C01786=1116.093,234.514,-69.767,-178.654,9.768,149.567
C01787=1116.097,234.266,-69.740,-178.657,9.765,149.567
C01788=1116.102,234.018,-69.713,-178.659,9.763,149.567
C01789=1116.106,233.768,-69.685,-178.662,9.761,149.567
C01790=1116.111,233.520,-69.658,-178.665,9.758,149.567
C01791=1116.115,233.272,-69.630,-178.667,9.755,149.567
C01792=1116.120,233.023,-69.603,-178.670,9.752,149.567
C01793=1116.124,232.774,-69.576,-178.673,9.749,149.567
C01794=1116.128,232.526,-69.549,-178.676,9.746,149.567
C01795=1116.132,232.278,-69.522,-178.680,9.743,149.568
C01796=1116.137,232.030,-69.495,-178.683,9.740,149.568
C01797=1116.141,231.781,-69.467,-178.685,9.737,149.568
C01798=1116.145,231.532,-69.440,-178.688,9.734,149.568
C01799=1116.150,231.284,-69.413,-178.691,9.732,149.568
C01800=1116.154,231.036,-69.386,-178.694,9.729,149.568
C01801=1116.158,230.787,-69.359,-178.697,9.726,149.568
C01802=1116.163,230.539,-69.332,-178.700,9.722,149.568
C01803=1116.167,230.290,-69.304,-178.703,9.719,149.568
C01804=1116.172,230.041,-69.277,-178.706,9.717,149.568
C01805=1116.176,229.793,-69.251,-178.710,9.713,149.568
C01806=1116.180,229.545,-69.224,-178.713,9.710,149.568
C01807=1116.185,229.296,-69.197,-178.715,9.707,149.568
C01808=1116.189,229.048,-69.170,-178.718,9.705,149.569
C01809=1116.193,228.799,-69.143,-178.722,9.701,149.569
C01810=1116.197,228.550,-69.116,-178.724,9.698,149.569
C01811=1116.202,228.302,-69.089,-178.727,9.695,149.569
C01812=1116.207,228.053,-69.061,-178.730,9.691,149.569
C01813=1116.211,227.805,-69.035,-178.733,9.688,149.569
C01814=1116.215,227.557,-69.008,-178.736,9.685,149.569
C01815=1116.220,227.308,-68.981,-178.739,9.683,149.569
C01816=1116.224,227.060,-68.954,-178.742,9.679,149.569
C01817=1116.228,226.847,-68.931,-178.744,9.677,149.569
C01818=1116.232,226.633,-68.908,-178.747,9.674,149.569
C01819=1116.236,226.420,-68.885,-178.749,9.671,149.569
C01820=1116.239,226.207,-68.862,-178.751,9.668,149.569
C01821=1116.243,225.993,-68.840,-178.754,9.665,149.569
C01822=1116.246,225.780,-68.816,-178.756,9.663,149.569
C01823=1116.251,225.567,-68.793,-178.758,9.660,149.569
C01824=1116.254,225.354,-68.770,-178.760,9.658,149.569
C01825=1116.258,225.105,-68.744,-178.763,9.655,149.569
C01826=1116.263,224.856,-68.717,-178.766,9.651,149.569
C01827=1116.267,224.608,-68.691,-178.769,9.648,149.569
C01828=1116.271,224.359,-68.663,-178.771,9.645,149.569
C01829=1116.276,224.110,-68.636,-178.774,9.642,149.568
C01830=1116.280,223.862,-68.610,-178.777,9.639,149.568
C01831=1116.285,223.613,-68.583,-178.780,9.636,149.569
C01832=1116.289,223.365,-68.557,-178.782,9.633,149.568
C01833=1116.294,223.116,-68.530,-178.785,9.630,149.568
C01834=1116.297,222.868,-68.504,-178.787,9.627,149.568
C01835=1116.302,222.619,-68.477,-178.790,9.623,149.568
C01836=1116.306,222.370,-68.451,-178.792,9.620,149.568
C01837=1116.311,222.122,-68.424,-178.795,9.617,149.568
C01838=1116.315,221.874,-68.398,-178.797,9.614,149.568
C01839=1116.320,221.624,-68.371,-178.800,9.611,149.568
C01840=1116.324,221.376,-68.345,-178.802,9.608,149.568
C01841=1116.328,221.128,-68.318,-178.804,9.604,149.568
C01842=1116.333,220.879,-68.292,-178.807,9.601,149.568
C01843=1116.337,220.630,-68.265,-178.809,9.598,149.568
C01844=1116.342,220.382,-68.240,-178.812,9.595,149.567
C01845=1116.346,220.134,-68.213,-178.814,9.592,149.567
C01846=1116.351,219.885,-68.187,-178.817,9.589,149.567
C01847=1116.355,219.637,-68.160,-178.819,9.586,149.567
C01848=1116.360,219.388,-68.134,-178.822,9.582,149.567
C01849=1116.364,219.140,-68.108,-178.823,9.580,149.567
C01850=1116.368,218.891,-68.082,-178.826,9.577,149.567
C01851=1116.373,218.642,-68.055,-178.829,9.574,149.567
C01852=1116.377,218.393,-68.029,-178.831,9.571,149.567
C01853=1116.381,218.145,-68.002,-178.833,9.567,149.567
C01854=1116.386,217.896,-67.976,-178.836,9.564,149.566
C01855=1116.390,217.648,-67.950,-178.838,9.562,149.566
C01856=1116.394,217.399,-67.924,-178.840,9.559,149.566
C01857=1116.399,217.150,-67.898,-178.842,9.555,149.566
C01858=1116.403,216.903,-67.871,-178.844,9.553,149.566
C01859=1116.408,216.654,-67.846,-178.847,9.550,149.566
C01860=1116.412,216.405,-67.819,-178.849,9.547,149.566
C01861=1116.417,216.157,-67.793,-178.851,9.543,149.566
C01862=1116.421,215.908,-67.767,-178.853,9.541,149.566
C01863=1116.425,215.659,-67.740,-178.856,9.538,149.566
C01864=1116.430,215.410,-67.714,-178.857,9.535,149.565
C01865=1116.434,215.162,-67.689,-178.860,9.532,149.565
C01866=1116.438,214.914,-67.662,-178.862,9.529,149.565
C01867=1116.443,214.665,-67.636,-178.864,9.526,149.565
C01868=1116.448,214.416,-67.610,-178.866,9.523,149.565
C01869=1116.452,214.167,-67.585,-178.868,9.521,149.565
C01870=1116.456,213.919,-67.558,-178.871,9.517,149.565
C01871=1116.461,213.670,-67.532,-178.872,9.515,149.564
C01872=1116.466,213.422,-67.506,-178.875,9.512,149.564
C01873=1116.469,213.209,-67.484,-178.877,9.509,149.564
C01874=1116.473,212.995,-67.461,-178.879,9.506,149.564
C01875=1116.476,212.782,-67.439,-178.881,9.504,149.564
C01876=1116.480,212.568,-67.418,-178.883,9.502,149.564
C01877=1116.484,212.355,-67.395,-178.885,9.498,149.564
C01878=1116.488,212.141,-67.373,-178.888,9.497,149.564
C01879=1116.492,211.928,-67.350,-178.890,9.494,149.564
C01880=1116.495,211.714,-67.328,-178.892,9.491,149.564
C01881=1116.500,211.466,-67.303,-178.895,9.488,149.564
C01882=1116.504,211.218,-67.277,-178.898,9.485,149.564
C01883=1116.509,210.968,-67.251,-178.900,9.482,149.564
C01884=1116.513,210.720,-67.225,-178.903,9.479,149.564
C01885=1116.518,210.472,-67.200,-178.906,9.476,149.564
C01886=1116.522,210.223,-67.174,-178.907,9.474,149.564
C01887=1116.527,209.974,-67.148,-178.910,9.471,149.564
C01888=1116.531,209.725,-67.122,-178.913,9.468,149.564
C01889=1116.536,209.477,-67.097,-178.915,9.465,149.564
C01890=1116.540,209.228,-67.071,-178.918,9.462,149.564
C01891=1116.544,208.979,-67.045,-178.921,9.459,149.564
C01892=1116.548,208.731,-67.020,-178.924,9.456,149.565
C01893=1116.553,208.483,-66.994,-178.927,9.454,149.565
C01894=1116.557,208.234,-66.969,-178.929,9.450,149.565
C01895=1116.562,207.985,-66.943,-178.932,9.448,149.565
C01896=1116.566,207.737,-66.917,-178.935,9.445,149.565
C01897=1116.571,207.488,-66.892,-178.938,9.442,149.565
C01898=1116.576,207.239,-66.865,-178.941,9.439,149.565
C01899=1116.580,206.991,-66.840,-178.943,9.436,149.565
C01900=1116.584,206.742,-66.815,-178.946,9.433,149.565
C01901=1116.588,206.493,-66.790,-178.949,9.431,149.565
C01902=1116.593,206.245,-66.764,-178.952,9.427,149.565
C01903=1116.597,205.996,-66.739,-178.955,9.425,149.565
C01904=1116.602,205.747,-66.713,-178.958,9.422,149.565
C01905=1116.607,205.499,-66.687,-178.961,9.419,149.566
C01906=1116.611,205.250,-66.662,-178.963,9.416,149.566
C01907=1116.615,205.001,-66.637,-178.966,9.413,149.566
C01908=1116.620,204.753,-66.611,-178.969,9.411,149.566
C01909=1116.624,204.504,-66.586,-178.972,9.408,149.566
C01910=1116.629,204.255,-66.561,-178.975,9.404,149.566
C01911=1116.634,204.006,-66.535,-178.978,9.401,149.566
C01912=1116.638,203.758,-66.509,-178.981,9.399,149.566
C01913=1116.643,203.509,-66.484,-178.984,9.396,149.566
C01914=1116.647,203.260,-66.460,-178.986,9.393,149.566
C01915=1116.651,203.012,-66.434,-178.989,9.390,149.566
C01916=1116.656,202.763,-66.408,-178.992,9.387,149.567
C01917=1116.660,202.514,-66.383,-178.995,9.384,149.567
C01918=1116.665,202.266,-66.358,-178.998,9.381,149.567
C01919=1116.669,202.016,-66.333,-179.001,9.378,149.567
C01920=1116.674,201.769,-66.308,-179.004,9.375,149.567
C01921=1116.678,201.520,-66.282,-179.007,9.372,149.567
C01922=1116.683,201.271,-66.258,-179.010,9.369,149.567
C01923=1116.687,201.022,-66.232,-179.013,9.366,149.567
C01924=1116.691,200.773,-66.208,-179.016,9.363,149.567
C01925=1116.696,200.525,-66.182,-179.019,9.360,149.567
C01926=1116.700,200.276,-66.157,-179.022,9.357,149.567
C01927=1116.705,200.028,-66.132,-179.025,9.354,149.568
C01928=1116.709,199.778,-66.107,-179.028,9.350,149.567
C01929=1116.713,199.565,-66.086,-179.031,9.348,149.568
C01930=1116.716,199.352,-66.064,-179.033,9.345,149.568
C01931=1116.721,199.139,-66.043,-179.036,9.343,149.568
C01932=1116.724,198.925,-66.021,-179.038,9.340,149.568
C01933=1116.728,198.711,-66.000,-179.041,9.337,149.568
C01934=1116.732,198.498,-65.979,-179.043,9.334,149.568
C01935=1116.736,198.284,-65.958,-179.046,9.332,149.568
C01936=1116.740,198.071,-65.936,-179.049,9.329,149.568
C01937=1116.745,197.822,-65.911,-179.052,9.326,149.568
C01938=1116.749,197.573,-65.886,-179.055,9.322,149.568
C01939=1116.753,197.325,-65.861,-179.058,9.319,149.568
C01940=1116.758,197.076,-65.836,-179.061,9.315,149.568
C01941=1116.763,196.827,-65.811,-179.064,9.313,149.568
C01942=1116.766,196.578,-65.786,-179.067,9.309,149.568
C01943=1116.772,196.330,-65.761,-179.069,9.306,149.568
C01944=1116.775,196.080,-65.737,-179.071,9.303,149.568
C01945=1116.781,195.832,-65.712,-179.073,9.300,149.568
C01946=1116.785,195.584,-65.687,-179.075,9.298,149.568
C01947=1116.789,195.335,-65.663,-179.077,9.295,149.568
C01948=1116.794,195.086,-65.638,-179.079,9.292,149.567
C01949=1116.798,194.837,-65.613,-179.081,9.289,149.567
C01950=1116.803,194.588,-65.589,-179.083,9.287,149.567
C01951=1116.807,194.340,-65.564,-179.085,9.284,149.567
C01952=1116.812,194.091,-65.539,-179.087,9.281,149.567
C01953=1116.816,193.842,-65.515,-179.089,9.279,149.567
C01954=1116.821,193.593,-65.490,-179.091,9.275,149.567
C01955=1116.825,193.345,-65.466,-179.093,9.273,149.567
C01956=1116.830,193.096,-65.441,-179.095,9.270,149.567
C01957=1116.834,192.847,-65.417,-179.097,9.267,149.566
C01958=1116.839,192.599,-65.391,-179.099,9.265,149.566
C01959=1116.843,192.350,-65.367,-179.101,9.262,149.566
C01960=1116.848,192.101,-65.342,-179.103,9.260,149.566
C01961=1116.852,191.852,-65.318,-179.106,9.256,149.566
C01962=1116.857,191.604,-65.293,-179.107,9.254,149.566
C01963=1116.861,191.354,-65.269,-179.110,9.251,149.566
C01964=1116.866,191.106,-65.244,-179.112,9.248,149.566
C01965=1116.871,190.857,-65.220,-179.114,9.245,149.566
C01966=1116.875,190.608,-65.195,-179.116,9.243,149.566
C01967=1116.880,190.360,-65.171,-179.119,9.240,149.566
C01968=1116.884,190.111,-65.147,-179.121,9.237,149.566
C01969=1116.889,189.862,-65.122,-179.123,9.234,149.566
C01970=1116.893,189.613,-65.098,-179.125,9.232,149.566
C01971=1116.898,189.365,-65.073,-179.127,9.229,149.566
C01972=1116.902,189.115,-65.049,-179.129,9.227,149.566
C01973=1116.906,188.867,-65.025,-179.132,9.223,149.566
C01974=1116.911,188.618,-65.000,-179.134,9.220,149.566
C01975=1116.916,188.370,-64.976,-179.136,9.218,149.566
C01976=1116.920,188.121,-64.952,-179.139,9.215,149.565
C01977=1116.925,187.871,-64.928,-179.141,9.213,149.565
C01978=1116.929,187.623,-64.904,-179.143,9.209,149.565
C01979=1116.935,187.374,-64.879,-179.146,9.206,149.565
C01980=1116.938,187.125,-64.854,-179.148,9.204,149.565
C01981=1116.943,186.877,-64.830,-179.150,9.201,149.565
C01982=1116.947,186.628,-64.806,-179.153,9.198,149.565
C01983=1116.952,186.380,-64.782,-179.155,9.195,149.565
C01984=1116.956,186.130,-64.758,-179.157,9.192,149.565
C01985=1116.961,185.917,-64.737,-179.159,9.190,149.565
C01986=1116.964,185.704,-64.716,-179.162,9.187,149.565
C01987=1116.968,185.489,-64.695,-179.163,9.185,149.565
C01988=1116.972,185.276,-64.674,-179.165,9.182,149.565
C01989=1116.976,185.062,-64.655,-179.168,9.180,149.565
C01990=1116.980,184.848,-64.633,-179.170,9.177,149.565
C01991=1116.984,184.634,-64.613,-179.172,9.175,149.565
C01992=1116.987,184.422,-64.592,-179.174,9.172,149.565
C01993=1116.993,184.173,-64.568,-179.176,9.169,149.565
C01994=1116.997,183.923,-64.544,-179.179,9.166,149.565
C01995=1117.001,183.675,-64.520,-179.182,9.163,149.565
C01996=1117.006,183.426,-64.496,-179.184,9.160,149.565
C01997=1117.010,183.177,-64.472,-179.187,9.157,149.565
C01998=1117.015,182.929,-64.448,-179.189,9.154,149.565
C01999=1117.020,182.680,-64.424,-179.192,9.151,149.565
C02000=1117.024,182.430,-64.400,-179.194,9.149,149.565
C02001=1117.028,182.182,-64.376,-179.196,9.146,149.565
C02002=1117.033,181.934,-64.352,-179.199,9.143,149.565
C02003=1117.037,181.685,-64.328,-179.201,9.139,149.565
C02004=1117.042,181.436,-64.304,-179.204,9.136,149.565
C02005=1117.046,181.187,-64.281,-179.207,9.133,149.565
C02006=1117.051,180.938,-64.256,-179.210,9.129,149.565
C02007=1117.056,180.689,-64.232,-179.212,9.126,149.565
C02008=1117.060,180.440,-64.208,-179.215,9.123,149.565
C02009=1117.065,180.191,-64.185,-179.217,9.120,149.564
C02010=1117.069,179.943,-64.161,-179.220,9.117,149.564
C02011=1117.074,179.694,-64.138,-179.222,9.114,149.564
C02012=1117.078,179.445,-64.114,-179.225,9.111,149.564
C02013=1117.083,179.196,-64.090,-179.227,9.108,149.564
C02014=1117.087,178.948,-64.066,-179.230,9.104,149.564
C02015=1117.092,178.699,-64.043,-179.231,9.102,149.564
C02016=1117.096,178.450,-64.018,-179.234,9.099,149.564
C02017=1117.101,178.201,-63.995,-179.236,9.096,149.564
C02018=1117.105,177.952,-63.972,-179.238,9.093,149.564
C02019=1117.110,177.703,-63.948,-179.240,9.090,149.564
C02020=1117.114,177.454,-63.924,-179.243,9.087,149.564
C02021=1117.119,177.205,-63.901,-179.244,9.084,149.563
C02022=1117.123,176.957,-63.877,-179.247,9.081,149.563
C02023=1117.128,176.708,-63.853,-179.249,9.078,149.563
C02024=1117.133,176.459,-63.830,-179.251,9.075,149.563
C02025=1117.137,176.210,-63.806,-179.253,9.072,149.563
C02026=1117.142,175.961,-63.783,-179.255,9.070,149.563
C02027=1117.147,175.712,-63.759,-179.257,9.066,149.563
C02028=1117.151,175.464,-63.735,-179.260,9.063,149.563
C02029=1117.156,175.215,-63.712,-179.262,9.061,149.563
C02030=1117.160,174.966,-63.688,-179.264,9.057,149.562
C02031=1117.165,174.717,-63.665,-179.266,9.054,149.562
C02032=1117.169,174.469,-63.642,-179.268,9.052,149.562
C02033=1117.173,174.220,-63.618,-179.271,9.049,149.562
C02034=1117.178,173.971,-63.595,-179.273,9.045,149.562
C02035=1117.183,173.722,-63.571,-179.275,9.042,149.562
C02036=1117.188,173.472,-63.548,-179.277,9.040,149.562
C02037=1117.192,173.224,-63.524,-179.279,9.036,149.562
C02038=1117.197,172.975,-63.501,-179.282,9.033,149.562
C02039=1117.201,172.726,-63.477,-179.284,9.031,149.562
C02040=1117.205,172.477,-63.455,-179.286,9.027,149.561
C02041=1117.210,172.263,-63.434,-179.288,9.025,149.561
C02042=1117.214,172.050,-63.414,-179.290,9.023,149.561
C02043=1117.217,171.836,-63.395,-179.292,9.019,149.561
C02044=1117.222,171.622,-63.374,-179.294,9.017,149.561
C02045=1117.226,171.409,-63.354,-179.296,9.014,149.561
C02046=1117.229,171.195,-63.335,-179.297,9.012,149.561
C02047=1117.233,170.981,-63.314,-179.299,9.010,149.561
C02048=1117.237,170.767,-63.294,-179.301,9.006,149.561
C02049=1117.242,170.518,-63.271,-179.303,9.004,149.561
C02050=1117.246,170.270,-63.248,-179.306,9.001,149.561
C02051=1117.251,170.021,-63.225,-179.308,8.997,149.561
C02052=1117.256,169.772,-63.202,-179.310,8.994,149.560
C02053=1117.260,169.523,-63.178,-179.312,8.992,149.560
C02054=1117.264,169.274,-63.155,-179.314,8.988,149.560
C02055=1117.269,169.025,-63.132,-179.317,8.985,149.560
C02056=1117.274,168.776,-63.109,-179.319,8.982,149.560
C02057=1117.279,168.527,-63.085,-179.321,8.980,149.560
C02058=1117.283,168.278,-63.063,-179.323,8.976,149.560
C02059=1117.288,168.030,-63.040,-179.326,8.973,149.560
C02060=1117.293,167.780,-63.017,-179.329,8.970,149.560
C02061=1117.297,167.532,-62.994,-179.330,8.967,149.560
C02062=1117.301,167.283,-62.971,-179.333,8.964,149.560
C02063=1117.306,167.034,-62.947,-179.335,8.961,149.559
C02064=1117.310,166.785,-62.925,-179.337,8.958,149.559
C02065=1117.315,166.537,-62.902,-179.340,8.955,149.559
C02066=1117.320,166.288,-62.878,-179.342,8.952,149.559
C02067=1117.324,166.038,-62.856,-179.344,8.949,149.559
C02068=1117.329,165.789,-62.833,-179.346,8.946,149.559
C02069=1117.334,165.540,-62.810,-179.348,8.942,149.559
C02070=1117.338,165.292,-62.787,-179.351,8.939,149.559
C02071=1117.343,165.043,-62.764,-179.353,8.936,149.559
C02072=1117.347,164.794,-62.742,-179.355,8.933,149.558
C02073=1117.352,164.545,-62.718,-179.357,8.930,149.558
C02074=1117.357,164.296,-62.695,-179.360,8.927,149.558
C02075=1117.361,164.048,-62.673,-179.362,8.924,149.558
C02076=1117.366,163.798,-62.650,-179.364,8.921,149.558
C02077=1117.370,163.549,-62.627,-179.366,8.917,149.558
C02078=1117.375,163.300,-62.604,-179.369,8.914,149.558
C02079=1117.379,163.051,-62.582,-179.371,8.912,149.558
C02080=1117.385,162.803,-62.559,-179.373,8.908,149.557
C02081=1117.389,162.554,-62.536,-179.375,8.905,149.557
C02082=1117.394,162.304,-62.513,-179.378,8.902,149.557
C02083=1117.397,162.056,-62.491,-179.380,8.898,149.557
C02084=1117.403,161.807,-62.468,-179.383,8.895,149.557
C02085=1117.407,161.558,-62.446,-179.385,8.892,149.557
C02086=1117.412,161.309,-62.422,-179.387,8.889,149.557
C02087=1117.417,161.060,-62.401,-179.389,8.885,149.557
C02088=1117.421,160.811,-62.377,-179.392,8.882,149.557
C02089=1117.425,160.562,-62.354,-179.393,8.879,149.556
C02090=1117.430,160.313,-62.332,-179.396,8.876,149.556
C02091=1117.435,160.065,-62.309,-179.398,8.873,149.556
C02092=1117.439,159.815,-62.287,-179.400,8.870,149.556
C02093=1117.444,159.566,-62.264,-179.403,8.867,149.556
C02094=1117.449,159.318,-62.242,-179.405,8.863,149.556
C02095=1117.453,159.069,-62.219,-179.408,8.860,149.556
C02096=1117.458,158.819,-62.197,-179.410,8.857,149.555
C02097=1117.462,158.605,-62.178,-179.412,8.853,149.555
C02098=1117.466,158.392,-62.158,-179.414,8.851,149.555
C02099=1117.470,158.178,-62.139,-179.415,8.848,149.555
C02100=1117.474,157.965,-62.120,-179.418,8.845,149.555
C02101=1117.478,157.750,-62.100,-179.419,8.843,149.555
C02102=1117.482,157.536,-62.081,-179.422,8.839,149.555
C02103=1117.485,157.323,-62.062,-179.423,8.837,149.555
C02104=1117.489,157.109,-62.043,-179.426,8.833,149.554
C02105=1117.494,156.859,-62.020,-179.428,8.830,149.554
C02106=1117.499,156.611,-61.998,-179.430,8.827,149.554
C02107=1117.503,156.362,-61.976,-179.433,8.824,149.554
C02108=1117.509,156.113,-61.954,-179.435,8.820,149.554
C02109=1117.513,155.864,-61.931,-179.437,8.817,149.554
C02110=1117.517,155.615,-61.909,-179.439,8.813,149.554
C02111=1117.523,155.366,-61.887,-179.441,8.810,149.553
C02112=1117.527,155.117,-61.864,-179.444,8.807,149.553
C02113=1117.531,154.868,-61.842,-179.446,8.803,149.553
C02114=1117.536,154.619,-61.820,-179.449,8.800,149.553
C02115=1117.541,154.370,-61.798,-179.451,8.797,149.553
C02116=1117.545,154.121,-61.775,-179.453,8.793,149.553
C02117=1117.549,153.872,-61.753,-179.455,8.790,149.553
C02118=1117.554,153.623,-61.731,-179.457,8.787,149.552
C02119=1117.559,153.374,-61.709,-179.460,8.782,149.552
C02120=1117.564,153.125,-61.687,-179.462,8.779,149.552
C02121=1117.568,152.876,-61.664,-179.465,8.776,149.552
C02122=1117.573,152.628,-61.643,-179.467,8.772,149.552
C02123=1117.577,152.378,-61.621,-179.469,8.769,149.551
C02124=1117.582,152.130,-61.599,-179.471,8.766,149.551
C02125=1117.587,151.880,-61.576,-179.473,8.762,149.551
C02126=1117.592,151.632,-61.555,-179.476,8.758,149.551
C02127=1117.596,151.382,-61.532,-179.478,8.754,149.551
C02128=1117.601,151.134,-61.511,-179.481,8.751,149.551
C02129=1117.605,150.884,-61.489,-179.483,8.748,149.550
C02130=1117.610,150.636,-61.467,-179.485,8.744,149.550
C02131=1117.615,150.386,-61.445,-179.487,8.741,149.550
C02132=1117.620,150.137,-61.423,-179.490,8.737,149.550
C02133=1117.624,149.888,-61.401,-179.492,8.734,149.550
C02134=1117.629,149.639,-61.379,-179.494,8.730,149.549
C02135=1117.634,149.390,-61.357,-179.496,8.727,149.549
C02136=1117.638,149.141,-61.335,-179.499,8.722,149.549
C02137=1117.643,148.892,-61.313,-179.501,8.719,149.549
C02138=1117.648,148.643,-61.292,-179.503,8.715,149.548
C02139=1117.652,148.395,-61.270,-179.505,8.712,149.548
C02140=1117.657,148.145,-61.248,-179.508,8.708,149.548
C02141=1117.662,147.897,-61.226,-179.510,8.704,149.548
C02142=1117.666,147.647,-61.204,-179.512,8.701,149.548
C02143=1117.671,147.399,-61.182,-179.515,8.697,149.547
C02144=1117.675,147.149,-61.160,-179.517,8.693,149.547
C02145=1117.680,146.900,-61.139,-179.519,8.690,149.547
C02146=1117.685,146.651,-61.118,-179.522,8.686,149.547
C02147=1117.689,146.402,-61.096,-179.524,8.682,149.547
C02148=1117.694,146.154,-61.074,-179.526,8.678,149.546
C02149=1117.699,145.905,-61.052,-179.528,8.675,149.546
C02150=1117.703,145.656,-61.030,-179.531,8.670,149.546
C02151=1117.709,145.406,-61.009,-179.533,8.667,149.545
C02152=1117.713,145.157,-60.987,-179.535,8.663,149.545
C02153=1117.717,144.944,-60.969,-179.536,8.661,149.545
C02154=1117.721,144.730,-60.950,-179.538,8.657,149.545
C02155=1117.724,144.515,-60.932,-179.539,8.654,149.544
C02156=1117.729,144.302,-60.913,-179.541,8.651,149.544
C02157=1117.733,144.087,-60.894,-179.542,8.649,149.544
C02158=1117.737,143.874,-60.876,-179.543,8.646,149.543
C02159=1117.742,143.659,-60.858,-179.545,8.643,149.543
C02160=1117.745,143.446,-60.839,-179.546,8.640,149.543
C02161=1117.750,143.197,-60.818,-179.548,8.636,149.542
C02162=1117.754,142.947,-60.796,-179.549,8.634,149.542
C02163=1117.759,142.698,-60.775,-179.551,8.630,149.542
C02164=1117.763,142.450,-60.754,-179.553,8.626,149.542
C02165=1117.768,142.200,-60.732,-179.554,8.623,149.541
C02166=1117.773,141.951,-60.711,-179.556,8.620,149.541
C02167=1117.778,141.702,-60.690,-179.557,8.617,149.540
C02168=1117.782,141.453,-60.668,-179.559,8.613,149.540
C02169=1117.787,141.204,-60.646,-179.561,8.609,149.540
C02170=1117.792,140.955,-60.626,-179.562,8.606,149.540
C02171=1117.796,140.707,-60.604,-179.564,8.603,149.539
C02172=1117.801,140.457,-60.583,-179.565,8.600,149.539
C02173=1117.806,140.208,-60.561,-179.567,8.596,149.538
C02174=1117.810,139.959,-60.540,-179.569,8.593,149.538
C02175=1117.815,139.710,-60.519,-179.570,8.589,149.538
C02176=1117.820,139.460,-60.497,-179.572,8.586,149.538
C02177=1117.825,139.212,-60.476,-179.574,8.583,149.537
C02178=1117.829,138.963,-60.455,-179.575,8.579,149.537
C02179=1117.834,138.714,-60.434,-179.577,8.576,149.537
C02180=1117.838,138.464,-60.412,-179.578,8.573,149.536
C02181=1117.843,138.216,-60.391,-179.580,8.569,149.536
C02182=1117.848,137.967,-60.370,-179.582,8.567,149.536
C02183=1117.853,137.718,-60.349,-179.583,8.563,149.535
C02184=1117.857,137.468,-60.327,-179.586,8.559,149.535
C02185=1117.861,137.220,-60.306,-179.587,8.556,149.535
C02186=1117.867,136.970,-60.285,-179.589,8.553,149.534
C02187=1117.872,136.721,-60.264,-179.591,8.549,149.534
C02188=1117.875,136.472,-60.243,-179.592,8.546,149.534
C02189=1117.880,136.223,-60.222,-179.594,8.543,149.534
C02190=1117.885,135.974,-60.200,-179.595,8.539,149.533
C02191=1117.890,135.725,-60.180,-179.597,8.536,149.533
C02192=1117.895,135.476,-60.159,-179.599,8.533,149.533
C02193=1117.900,135.227,-60.137,-179.600,8.529,149.532
C02194=1117.904,134.978,-60.116,-179.602,8.526,149.532
C02195=1117.909,134.729,-60.095,-179.604,8.522,149.532
C02196=1117.914,134.480,-60.074,-179.605,8.519,149.531
C02197=1117.918,134.231,-60.053,-179.607,8.516,149.531
C02198=1117.923,133.982,-60.032,-179.609,8.513,149.531
C02199=1117.928,133.733,-60.012,-179.610,8.509,149.530
C02200=1117.932,133.483,-59.990,-179.612,8.506,149.530
C02201=1117.937,133.234,-59.969,-179.614,8.503,149.530
C02202=1117.942,132.985,-59.949,-179.616,8.500,149.530
C02203=1117.947,132.736,-59.928,-179.617,8.496,149.529
C02204=1117.951,132.487,-59.907,-179.619,8.493,149.529
C02205=1117.956,132.238,-59.886,-179.621,8.489,149.529
C02206=1117.961,131.989,-59.865,-179.623,8.486,149.528
C02207=1117.966,131.740,-59.844,-179.624,8.483,149.528
C02208=1117.970,131.490,-59.824,-179.626,8.479,149.528
C02209=1117.975,131.250,-59.803,-179.628,8.477,149.528
C02210=1117.979,131.010,-59.783,-179.629,8.473,149.527
C02211=1117.984,130.769,-59.763,-179.631,8.470,149.527
C02212=1117.989,130.528,-59.743,-179.633,8.467,149.527
C02213=1117.993,130.288,-59.723,-179.634,8.464,149.527
C02214=1117.997,130.047,-59.703,-179.636,8.460,149.526
C02215=1118.002,129.806,-59.683,-179.637,8.457,149.526
C02216=1118.007,129.566,-59.663,-179.639,8.454,149.526
C02217=1118.012,129.317,-59.642,-179.641,8.450,149.526
C02218=1118.017,129.068,-59.622,-179.642,8.447,149.525
C02219=1118.021,128.818,-59.601,-179.644,8.444,149.525
C02220=1118.025,128.570,-59.580,-179.646,8.440,149.525
C02221=1118.030,128.321,-59.559,-179.648,8.438,149.524
C02222=1118.034,128.072,-59.538,-179.650,8.434,149.524
C02223=1118.040,127.823,-59.517,-179.652,8.430,149.524
C02224=1118.044,127.574,-59.497,-179.653,8.427,149.524
C02225=1118.049,127.324,-59.476,-179.655,8.424,149.523
C02226=1118.054,127.075,-59.456,-179.657,8.420,149.523
C02227=1118.058,126.826,-59.436,-179.658,8.417,149.523
C02228=1118.063,126.577,-59.415,-179.660,8.414,149.522
C02229=1118.068,126.355,-59.397,-179.662,8.411,149.522
C02230=1118.071,126.132,-59.378,-179.664,8.408,149.522
C02231=1118.076,125.909,-59.360,-179.665,8.405,149.522
C02232=1118.080,125.687,-59.342,-179.666,8.402,149.521
C02233=1118.084,125.464,-59.324,-179.668,8.398,149.521
C02234=1118.089,125.241,-59.305,-179.670,8.396,149.521
C02235=1118.093,125.019,-59.287,-179.671,8.393,149.521
C02236=1118.097,124.796,-59.269,-179.673,8.390,149.520
C02237=1118.101,124.547,-59.248,-179.675,8.387,149.520
C02238=1118.107,124.298,-59.227,-179.677,8.383,149.520
C02239=1118.111,124.049,-59.207,-179.678,8.379,149.520
C02240=1118.115,123.800,-59.187,-179.680,8.377,149.519
C02241=1118.121,123.550,-59.166,-179.682,8.373,149.519
C02242=1118.125,123.301,-59.146,-179.684,8.370,149.519
C02243=1118.130,123.052,-59.126,-179.685,8.366,149.518
C02244=1118.134,122.803,-59.105,-179.687,8.363,149.518
C02245=1118.139,122.554,-59.084,-179.689,8.359,149.518
C02246=1118.144,122.305,-59.064,-179.690,8.357,149.518
C02247=1118.149,122.056,-59.045,-179.693,8.353,149.518
C02248=1118.154,121.807,-59.024,-179.694,8.349,149.517
C02249=1118.159,121.558,-59.003,-179.696,8.346,149.517
C02250=1118.163,121.309,-58.983,-179.698,8.343,149.517
C02251=1118.168,121.059,-58.963,-179.700,8.340,149.516
C02252=1118.172,120.810,-58.943,-179.701,8.336,149.516
C02253=1118.177,120.561,-58.923,-179.703,8.332,149.516
C02254=1118.182,120.311,-58.902,-179.705,8.330,149.516
C02255=1118.187,120.062,-58.882,-179.707,8.326,149.515
C02256=1118.191,119.814,-58.862,-179.709,8.322,149.515
C02257=1118.196,119.564,-58.842,-179.711,8.319,149.515
C02258=1118.201,119.316,-58.822,-179.712,8.316,149.514
C02259=1118.206,119.066,-58.801,-179.714,8.313,149.514
C02260=1118.211,118.817,-58.781,-179.716,8.309,149.514
C02261=1118.215,118.568,-58.761,-179.718,8.305,149.514
C02262=1118.220,118.318,-58.741,-179.719,8.302,149.513
C02263=1118.225,118.069,-58.721,-179.721,8.299,149.513
C02264=1118.229,117.820,-58.701,-179.723,8.295,149.513
C02265=1118.234,117.606,-58.684,-179.725,8.293,149.513
C02266=1118.238,117.392,-58.666,-179.726,8.290,149.512
C02267=1118.242,117.178,-58.650,-179.728,8.286,149.512
C02268=1118.246,116.963,-58.632,-179.729,8.283,149.512
C02269=1118.250,116.750,-58.615,-179.731,8.281,149.512
C02270=1118.254,116.535,-58.598,-179.732,8.278,149.511
C02271=1118.258,116.321,-58.581,-179.734,8.274,149.511
C02272=1118.262,116.107,-58.563,-179.736,8.272,149.511
C02273=1118.267,115.858,-58.544,-179.738,8.268,149.511
C02274=1118.271,115.609,-58.523,-179.739,8.266,149.510
C02275=1118.276,115.360,-58.504,-179.741,8.262,149.510
C02276=1118.281,115.111,-58.484,-179.743,8.258,149.510
C02277=1118.286,114.861,-58.464,-179.745,8.255,149.510
C02278=1118.290,114.612,-58.444,-179.747,8.251,149.509
C02279=1118.295,114.363,-58.424,-179.749,8.247,149.509
C02280=1118.300,114.114,-58.405,-179.750,8.245,149.509
C02281=1118.305,113.865,-58.384,-179.752,8.241,149.508
C02282=1118.309,113.615,-58.365,-179.754,8.237,149.508
C02283=1118.315,113.367,-58.345,-179.756,8.234,149.508
C02284=1118.319,113.118,-58.325,-179.758,8.230,149.508
C02285=1118.324,112.868,-58.305,-179.759,8.227,149.507
C02286=1118.329,112.618,-58.286,-179.761,8.224,149.507
C02287=1118.334,112.370,-58.266,-179.763,8.220,149.507
C02288=1118.338,112.121,-58.246,-179.765,8.217,149.506
C02289=1118.343,111.871,-58.226,-179.767,8.213,149.506
C02290=1118.348,111.621,-58.207,-179.769,8.209,149.506
C02291=1118.353,111.373,-58.187,-179.771,8.206,149.506
C02292=1118.358,111.124,-58.167,-179.772,8.203,149.505
C02293=1118.362,110.874,-58.147,-179.774,8.198,149.505
C02294=1118.368,110.625,-58.128,-179.776,8.195,149.505
C02295=1118.372,110.376,-58.108,-179.779,8.191,149.504
C02296=1118.377,110.127,-58.088,-179.781,8.188,149.504
C02297=1118.382,109.878,-58.069,-179.783,8.184,149.504
C02298=1118.386,109.629,-58.050,-179.785,8.180,149.504
C02299=1118.391,109.379,-58.030,-179.787,8.177,149.504
C02300=1118.396,109.131,-58.010,-179.790,8.172,149.503
C02301=1118.401,108.881,-57.990,-179.792,8.169,149.503
C02302=1118.406,108.632,-57.971,-179.794,8.165,149.503
C02303=1118.411,108.383,-57.951,-179.796,8.161,149.502
C02304=1118.415,108.134,-57.932,-179.798,8.157,149.502
C02305=1118.420,107.884,-57.913,-179.801,8.154,149.502
C02306=1118.425,107.635,-57.893,-179.803,8.150,149.502
C02307=1118.430,107.386,-57.874,-179.805,8.145,149.501
C02308=1118.434,107.136,-57.855,-179.807,8.142,149.501
C02309=1118.439,106.887,-57.835,-179.809,8.138,149.501
C02310=1118.444,106.638,-57.816,-179.811,8.135,149.500
C02311=1118.449,106.389,-57.796,-179.813,8.130,149.500
C02312=1118.453,106.140,-57.777,-179.815,8.127,149.500
C02313=1118.458,105.890,-57.758,-179.817,8.123,149.500
C02314=1118.463,105.641,-57.738,-179.819,8.119,149.499
C02315=1118.468,105.392,-57.719,-179.821,8.116,149.499
C02316=1118.473,105.143,-57.700,-179.823,8.111,149.499
C02317=1118.477,104.894,-57.680,-179.825,8.108,149.498
C02318=1118.483,104.645,-57.661,-179.827,8.104,149.498
C02319=1118.487,104.395,-57.642,-179.829,8.100,149.498
C02320=1118.491,104.146,-57.622,-179.831,8.096,149.497
C02321=1118.496,103.931,-57.606,-179.833,8.093,149.497
C02322=1118.500,103.717,-57.590,-179.835,8.089,149.497
C02323=1118.504,103.503,-57.573,-179.836,8.087,149.497
C02324=1118.508,103.289,-57.557,-179.838,8.083,149.496
C02325=1118.513,103.074,-57.540,-179.839,8.080,149.496
C02326=1118.517,102.860,-57.524,-179.841,8.077,149.496
C02327=1118.521,102.646,-57.507,-179.843,8.073,149.495
C02328=1118.525,102.432,-57.491,-179.844,8.070,149.495
C02329=1118.530,102.182,-57.472,-179.846,8.066,149.495
C02330=1118.534,101.934,-57.453,-179.848,8.063,149.495
C02331=1118.539,101.684,-57.433,-179.850,8.058,149.494
C02332=1118.544,101.436,-57.414,-179.852,8.054,149.494
C02333=1118.549,101.185,-57.396,-179.854,8.050,149.493
C02334=1118.554,100.937,-57.376,-179.855,8.047,149.493
C02335=1118.558,100.687,-57.357,-179.857,8.043,149.493
C02336=1118.563,100.438,-57.338,-179.859,8.039,149.492
C02337=1118.568,100.189,-57.320,-179.861,8.035,149.492
C02338=1118.573,99.940,-57.300,-179.862,8.031,149.492
C02339=1118.578,99.691,-57.282,-179.865,8.027,149.491
C02340=1118.583,99.441,-57.263,-179.867,8.023,149.491
C02341=1118.587,99.192,-57.244,-179.868,8.019,149.490
C02342=1118.592,98.943,-57.224,-179.870,8.015,149.490
C02343=1118.597,98.694,-57.206,-179.871,8.012,149.490
C02344=1118.602,98.444,-57.187,-179.873,8.008,149.489
C02345=1118.607,98.195,-57.169,-179.875,8.004,149.489
C02346=1118.612,97.946,-57.149,-179.877,8.000,149.488
C02347=1118.616,97.697,-57.130,-179.878,7.996,149.488
C02348=1118.622,97.447,-57.112,-179.880,7.993,149.488
C02349=1118.626,97.198,-57.093,-179.881,7.989,149.487
C02350=1118.631,96.949,-57.075,-179.883,7.985,149.487
C02351=1118.636,96.700,-57.055,-179.885,7.981,149.487
C02352=1118.640,96.450,-57.037,-179.887,7.977,149.486
C02353=1118.646,96.201,-57.018,-179.888,7.973,149.486
C02354=1118.650,95.951,-56.999,-179.890,7.970,149.485
C02355=1118.654,95.703,-56.981,-179.891,7.966,149.485
C02356=1118.660,95.453,-56.962,-179.893,7.962,149.484
C02357=1118.664,95.204,-56.943,-179.895,7.958,149.484
C02358=1118.670,94.955,-56.925,-179.896,7.954,149.484
C02359=1118.674,94.706,-56.906,-179.898,7.950,149.483
C02360=1118.679,94.456,-56.887,-179.899,7.946,149.483
C02361=1118.684,94.207,-56.868,-179.901,7.942,149.482
C02362=1118.689,93.958,-56.850,-179.903,7.938,149.482
C02363=1118.693,93.708,-56.832,-179.904,7.935,149.481
C02364=1118.699,93.459,-56.813,-179.906,7.931,149.481
C02365=1118.704,93.210,-56.795,-179.907,7.927,149.480
C02366=1118.708,92.961,-56.776,-179.909,7.923,149.480
C02367=1118.713,92.711,-56.757,-179.911,7.919,149.480
C02368=1118.718,92.462,-56.739,-179.912,7.915,149.479
C02369=1118.722,92.213,-56.720,-179.913,7.911,149.479
C02370=1118.728,91.963,-56.701,-179.914,7.908,149.478
C02371=1118.733,91.714,-56.683,-179.916,7.904,149.478
C02372=1118.737,91.465,-56.664,-179.918,7.900,149.477
C02373=1118.742,91.216,-56.646,-179.919,7.896,149.477
C02374=1118.747,90.966,-56.628,-179.921,7.892,149.476
C02375=1118.752,90.717,-56.610,-179.922,7.888,149.476
C02376=1118.756,90.468,-56.591,-179.923,7.884,149.475
C02377=1118.760,90.253,-56.575,-179.925,7.881,149.475
C02378=1118.765,90.040,-56.560,-179.926,7.878,149.475
C02379=1118.770,89.825,-56.544,-179.927,7.874,149.474
C02380=1118.773,89.611,-56.527,-179.928,7.871,149.474
C02381=1118.777,89.396,-56.512,-179.929,7.868,149.473
C02382=1118.781,89.182,-56.496,-179.931,7.864,149.473
C02383=1118.785,88.967,-56.481,-179.932,7.861,149.473
C02384=1118.789,88.753,-56.465,-179.933,7.858,149.472
C02385=1118.794,88.504,-56.447,-179.935,7.854,149.472
C02386=1118.800,88.254,-56.428,-179.936,7.850,149.471
C02387=1118.805,88.005,-56.410,-179.937,7.847,149.471
C02388=1118.810,87.756,-56.392,-179.938,7.843,149.470
C02389=1118.814,87.506,-56.374,-179.940,7.839,149.470
C02390=1118.819,87.258,-56.355,-179.941,7.835,149.469
C02391=1118.823,87.008,-56.337,-179.943,7.831,149.469
C02392=1118.828,86.759,-56.319,-179.944,7.828,149.468
C02393=1118.834,86.510,-56.300,-179.945,7.823,149.468
C02394=1118.838,86.260,-56.282,-179.946,7.819,149.467
C02395=1118.843,86.011,-56.264,-179.947,7.816,149.467
C02396=1118.848,85.762,-56.246,-179.948,7.812,149.466
C02397=1118.853,85.512,-56.228,-179.950,7.808,149.466
C02398=1118.858,85.263,-56.210,-179.952,7.804,149.465
C02399=1118.862,85.013,-56.192,-179.952,7.801,149.465
C02400=1118.867,84.764,-56.174,-179.954,7.797,149.464
C02401=1118.872,84.515,-56.156,-179.955,7.793,149.464
C02402=1118.877,84.266,-56.138,-179.956,7.789,149.463
C02403=1118.882,84.017,-56.120,-179.957,7.786,149.463
C02404=1118.887,83.767,-56.102,-179.958,7.781,149.462
C02405=1118.892,83.518,-56.084,-179.959,7.778,149.462
C02406=1118.897,83.268,-56.065,-179.961,7.774,149.461
C02407=1118.902,83.019,-56.047,-179.962,7.770,149.460
C02408=1118.907,82.770,-56.029,-179.963,7.767,149.460
C02409=1118.912,82.521,-56.011,-179.964,7.763,149.459
C02410=1118.916,82.271,-55.993,-179.965,7.759,149.459
C02411=1118.921,82.022,-55.975,-179.966,7.755,149.458
C02412=1118.926,81.773,-55.957,-179.968,7.751,149.458
C02413=1118.931,81.524,-55.939,-179.968,7.748,149.457
C02414=1118.936,81.275,-55.921,-179.970,7.744,149.457
C02415=1118.940,81.024,-55.904,-179.971,7.740,149.456
C02416=1118.945,80.775,-55.886,-179.972,7.737,149.456
C02417=1118.950,80.526,-55.868,-179.973,7.732,149.455
C02418=1118.955,80.277,-55.850,-179.974,7.729,149.455
C02419=1118.960,80.028,-55.832,-179.975,7.725,149.454
C02420=1118.965,79.779,-55.814,-179.976,7.722,149.454
C02421=1118.970,79.529,-55.797,-179.977,7.717,149.453
C02422=1118.975,79.280,-55.779,-179.978,7.714,149.453
C02423=1118.980,79.030,-55.761,-179.979,7.710,149.452
C02424=1118.985,78.781,-55.743,-179.980,7.707,149.451
C02425=1118.989,78.532,-55.725,-179.982,7.703,149.451
C02426=1118.995,78.282,-55.708,-179.982,7.699,149.450
C02427=1119.000,78.033,-55.690,-179.984,7.695,149.450
C02428=1119.004,77.784,-55.672,-179.984,7.692,149.449
C02429=1119.009,77.535,-55.654,-179.986,7.688,149.449
C02430=1119.014,77.285,-55.637,-179.986,7.684,149.448
C02431=1119.019,77.036,-55.619,-179.987,7.681,149.447
C02432=1119.023,76.786,-55.601,-179.988,7.677,149.447
C02433=1119.028,76.572,-55.586,-179.989,7.674,149.446
C02434=1119.032,76.357,-55.570,-179.991,7.670,149.446
C02435=1119.036,76.143,-55.555,-179.992,7.667,149.446
C02436=1119.040,75.929,-55.541,-179.993,7.664,149.445
C02437=1119.044,75.714,-55.525,-179.994,7.660,149.445
C02438=1119.048,75.500,-55.510,-179.995,7.657,149.444
C02439=1119.053,75.286,-55.495,-179.997,7.653,149.444
C02440=1119.057,75.071,-55.479,-179.998,7.650,149.443
C02441=1119.062,74.821,-55.462,-179.999,7.646,149.443
C02442=1119.067,74.572,-55.445,179.999,7.642,149.443
C02443=1119.071,74.323,-55.427,179.997,7.638,149.442
C02444=1119.077,74.073,-55.410,179.996,7.634,149.442
C02445=1119.082,73.824,-55.392,179.995,7.630,149.441
C02446=1119.086,73.575,-55.375,179.993,7.626,149.441
C02447=1119.091,73.325,-55.357,179.992,7.622,149.440
C02448=1119.096,73.076,-55.340,179.990,7.618,149.440
C02449=1119.101,72.826,-55.322,179.989,7.615,149.439
C02450=1119.105,72.578,-55.304,179.988,7.611,149.439
C02451=1119.111,72.328,-55.287,179.987,7.606,149.438
C02452=1119.115,72.079,-55.269,179.985,7.602,149.438
C02453=1119.121,71.830,-55.252,179.984,7.599,149.437
C02454=1119.125,71.581,-55.235,179.982,7.595,149.437
C02455=1119.131,71.331,-55.218,179.981,7.590,149.436
C02456=1119.136,71.082,-55.200,179.979,7.587,149.436
C02457=1119.140,70.832,-55.183,179.978,7.583,149.435
C02458=1119.145,70.582,-55.166,179.977,7.578,149.435
C02459=1119.150,70.333,-55.148,179.975,7.574,149.434
C02460=1119.155,70.084,-55.131,179.974,7.571,149.434
C02461=1119.160,69.835,-55.113,179.972,7.567,149.433
C02462=1119.165,69.585,-55.096,179.971,7.562,149.433
C02463=1119.170,69.336,-55.079,179.969,7.558,149.432
C02464=1119.175,69.087,-55.061,179.968,7.555,149.432
C02465=1119.180,68.837,-55.044,179.967,7.551,149.431
C02466=1119.184,68.588,-55.027,179.966,7.547,149.431
C02467=1119.189,68.338,-55.010,179.964,7.543,149.430
C02468=1119.194,68.089,-54.993,179.963,7.539,149.430
C02469=1119.199,67.840,-54.975,179.961,7.535,149.429
C02470=1119.205,67.591,-54.958,179.960,7.531,149.429
C02471=1119.209,67.341,-54.941,179.959,7.527,149.428
C02472=1119.214,67.092,-54.923,179.957,7.523,149.428
C02473=1119.218,66.842,-54.907,179.956,7.519,149.427
C02474=1119.224,66.593,-54.889,179.954,7.515,149.427
C02475=1119.228,66.343,-54.873,179.953,7.511,149.426
C02476=1119.234,66.095,-54.855,179.951,7.507,149.426
C02477=1119.238,65.845,-54.838,179.951,7.503,149.425
C02478=1119.243,65.595,-54.821,179.949,7.499,149.425
C02479=1119.248,65.346,-54.804,179.948,7.496,149.424
C02480=1119.253,65.096,-54.787,179.947,7.491,149.424
C02481=1119.258,64.848,-54.770,179.945,7.487,149.423
C02482=1119.263,64.598,-54.753,179.943,7.483,149.423
C02483=1119.268,64.349,-54.736,179.942,7.479,149.422
C02484=1119.273,64.099,-54.719,179.941,7.475,149.422
C02485=1119.277,63.849,-54.702,179.939,7.471,149.421
C02486=1119.283,63.600,-54.685,179.938,7.467,149.421
C02487=1119.287,63.351,-54.668,179.937,7.463,149.420
C02488=1119.292,63.102,-54.651,179.936,7.460,149.420
C02489=1119.297,62.887,-54.637,179.934,7.456,149.419
C02490=1119.301,62.673,-54.622,179.934,7.453,149.419
C02491=1119.305,62.458,-54.608,179.932,7.449,149.418
C02492=1119.309,62.244,-54.593,179.931,7.446,149.418
C02493=1119.314,62.029,-54.579,179.930,7.442,149.417
C02494=1119.318,61.815,-54.564,179.929,7.439,149.417
C02495=1119.322,61.600,-54.550,179.928,7.435,149.417
C02496=1119.326,61.385,-54.535,179.927,7.432,149.416
C02497=1119.331,61.135,-54.518,179.925,7.428,149.416
C02498=1119.337,60.886,-54.502,179.924,7.424,149.415
C02499=1119.341,60.637,-54.485,179.922,7.420,149.415
C02500=1119.346,60.387,-54.468,179.921,7.416,149.414
C02501=1119.352,60.138,-54.451,179.920,7.412,149.414
C02502=1119.356,59.889,-54.435,179.919,7.408,149.413
C02503=1119.360,59.639,-54.418,179.917,7.404,149.412
C02504=1119.366,59.390,-54.401,179.916,7.400,149.412
C02505=1119.371,59.141,-54.384,179.914,7.396,149.411
C02506=1119.375,58.891,-54.368,179.913,7.392,149.411
C02507=1119.381,58.642,-54.351,179.912,7.388,149.410
C02508=1119.386,58.393,-54.334,179.911,7.384,149.410
C02509=1119.390,58.143,-54.318,179.910,7.380,149.409
C02510=1119.396,57.894,-54.301,179.908,7.376,149.409
C02511=1119.400,57.645,-54.284,179.907,7.372,149.408
C02512=1119.405,57.395,-54.267,179.906,7.368,149.408
C02513=1119.410,57.146,-54.251,179.904,7.364,149.407
C02514=1119.415,56.896,-54.234,179.903,7.360,149.407
C02515=1119.420,56.646,-54.218,179.901,7.356,149.406
C02516=1119.425,56.398,-54.201,179.900,7.351,149.406
C02517=1119.430,56.148,-54.184,179.899,7.348,149.405
C02518=1119.435,55.899,-54.168,179.898,7.344,149.405
C02519=1119.440,55.649,-54.152,179.897,7.340,149.404
C02520=1119.445,55.399,-54.135,179.896,7.336,149.403
C02521=1119.450,55.151,-54.119,179.894,7.332,149.403
C02522=1119.455,54.901,-54.102,179.893,7.328,149.402
C02523=1119.460,54.652,-54.085,179.891,7.324,149.402
C02524=1119.465,54.402,-54.069,179.890,7.319,149.401
C02525=1119.470,54.153,-54.053,179.889,7.316,149.401
C02526=1119.474,53.904,-54.036,179.888,7.311,149.400
C02527=1119.479,53.654,-54.019,179.887,7.308,149.400
C02528=1119.485,53.404,-54.004,179.886,7.304,149.399
C02529=1119.489,53.155,-53.987,179.884,7.300,149.399
C02530=1119.494,52.906,-53.971,179.883,7.296,149.398
C02531=1119.499,52.656,-53.955,179.881,7.292,149.398
C02532=1119.504,52.407,-53.938,179.880,7.287,149.397
C02533=1119.510,52.158,-53.921,179.879,7.283,149.396
C02534=1119.515,51.908,-53.906,179.878,7.279,149.396
C02535=1119.519,51.659,-53.889,179.877,7.275,149.395
C02536=1119.525,51.409,-53.873,179.875,7.271,149.395
C02537=1119.529,51.160,-53.857,179.875,7.267,149.394
C02538=1119.534,50.910,-53.840,179.873,7.264,149.394
C02539=1119.539,50.661,-53.824,179.872,7.259,149.393
C02540=1119.544,50.411,-53.808,179.870,7.255,149.393
C02541=1119.549,50.162,-53.792,179.869,7.251,149.392
C02542=1119.553,49.912,-53.775,179.868,7.247,149.391
C02543=1119.559,49.664,-53.759,179.867,7.243,149.391
C02544=1119.563,49.414,-53.743,179.865,7.238,149.390
C02545=1119.568,49.199,-53.729,179.865,7.235,149.390
C02546=1119.573,48.985,-53.715,179.864,7.232,149.389
C02547=1119.577,48.770,-53.701,179.863,7.228,149.389
C02548=1119.581,48.555,-53.687,179.862,7.225,149.388
C02549=1119.585,48.341,-53.674,179.860,7.221,149.388
C02550=1119.590,48.126,-53.659,179.859,7.218,149.387
C02551=1119.594,47.911,-53.645,179.859,7.214,149.387
C02552=1119.598,47.696,-53.632,179.857,7.210,149.386
C02553=1119.603,47.448,-53.616,179.856,7.206,149.386
C02554=1119.608,47.197,-53.600,179.855,7.203,149.385
C02555=1119.613,46.949,-53.584,179.854,7.199,149.385
C02556=1119.618,46.699,-53.568,179.852,7.195,149.384
C02557=1119.623,46.450,-53.551,179.851,7.190,149.384
C02558=1119.628,46.200,-53.536,179.850,7.186,149.383
C02559=1119.633,45.950,-53.520,179.849,7.182,149.383
C02560=1119.638,45.701,-53.504,179.848,7.178,149.382
C02561=1119.643,45.451,-53.488,179.847,7.174,149.381
C02562=1119.648,45.203,-53.471,179.845,7.170,149.381
C02563=1119.652,44.953,-53.456,179.844,7.165,149.380
C02564=1119.658,44.703,-53.440,179.844,7.162,149.379
C02565=1119.663,44.455,-53.424,179.842,7.158,149.379
C02566=1119.668,44.205,-53.408,179.841,7.154,149.378
C02567=1119.673,43.955,-53.393,179.840,7.149,149.378
C02568=1119.677,43.706,-53.376,179.839,7.145,149.377
C02569=1119.683,43.456,-53.360,179.837,7.141,149.377
C02570=1119.688,43.207,-53.345,179.836,7.137,149.376
C02571=1119.693,42.957,-53.329,179.835,7.132,149.375
C02572=1119.697,42.708,-53.313,179.834,7.128,149.375
C02573=1119.703,42.459,-53.298,179.832,7.124,149.374
C02574=1119.707,42.209,-53.282,179.831,7.120,149.374
C02575=1119.713,41.959,-53.266,179.831,7.116,149.373
C02576=1119.718,41.711,-53.250,179.829,7.112,149.373
C02577=1119.723,41.460,-53.234,179.828,7.108,149.372
C02578=1119.727,41.211,-53.219,179.827,7.104,149.371
C02579=1119.733,40.962,-53.203,179.826,7.100,149.371
C02580=1119.738,40.712,-53.187,179.825,7.095,149.370
C02581=1119.743,40.462,-53.172,179.824,7.091,149.370
C02582=1119.748,40.214,-53.155,179.822,7.087,149.369
C02583=1119.752,39.964,-53.140,179.821,7.083,149.368
C02584=1119.757,39.714,-53.124,179.820,7.078,149.368
C02585=1119.763,39.465,-53.109,179.819,7.074,149.367
C02586=1119.768,39.215,-53.093,179.818,7.071,149.367
C02587=1119.772,38.966,-53.078,179.817,7.067,149.366
C02588=1119.778,38.716,-53.062,179.816,7.062,149.365
C02589=1119.783,38.467,-53.047,179.815,7.058,149.365
C02590=1119.788,38.217,-53.031,179.814,7.054,149.364
C02591=1119.792,37.968,-53.016,179.813,7.049,149.363
C02592=1119.798,37.719,-52.999,179.811,7.046,149.363
C02593=1119.803,37.470,-52.984,179.810,7.041,149.362
C02594=1119.807,37.220,-52.968,179.809,7.037,149.362
C02595=1119.812,36.971,-52.953,179.808,7.033,149.361
C02596=1119.818,36.721,-52.937,179.807,7.028,149.360
C02597=1119.823,36.472,-52.922,179.806,7.024,149.360
C02598=1119.827,36.222,-52.906,179.806,7.020,149.359
C02599=1119.833,35.973,-52.891,179.805,7.016,149.358
C02600=1119.838,35.723,-52.875,179.803,7.012,149.358
C02601=1119.842,35.508,-52.863,179.802,7.008,149.357
C02602=1119.846,35.294,-52.850,179.801,7.005,149.357
C02603=1119.851,35.079,-52.836,179.801,7.001,149.356
C02604=1119.855,34.864,-52.823,179.799,6.997,149.356
C02605=1119.859,34.649,-52.809,179.799,6.994,149.355
C02606=1119.864,34.434,-52.796,179.798,6.990,149.354
C02607=1119.868,34.219,-52.783,179.797,6.986,149.354
C02608=1119.873,34.005,-52.769,179.796,6.983,149.353
C02609=1119.877,33.756,-52.754,179.795,6.979,149.353
C02610=1119.883,33.506,-52.739,179.794,6.975,149.352
C02611=1119.888,33.257,-52.724,179.793,6.970,149.352
C02612=1119.892,33.007,-52.708,179.791,6.966,149.351
C02613=1119.897,32.758,-52.693,179.790,6.962,149.350
C02614=1119.902,32.508,-52.678,179.789,6.957,149.350
C02615=1119.908,32.259,-52.662,179.788,6.953,149.349
C02616=1119.912,32.010,-52.647,179.787,6.949,149.348
C02617=1119.918,31.760,-52.632,179.786,6.944,149.348
C02618=1119.922,31.510,-52.617,179.785,6.940,149.347
C02619=1119.927,31.260,-52.601,179.784,6.936,149.346
C02620=1119.932,31.011,-52.586,179.783,6.931,149.346
C02621=1119.938,30.761,-52.572,179.782,6.927,149.345
C02622=1119.942,30.512,-52.557,179.782,6.923,149.344
C02623=1119.948,30.263,-52.541,179.781,6.919,149.344
C02624=1119.953,30.014,-52.526,179.780,6.915,149.343
C02625=1119.958,29.764,-52.511,179.779,6.910,149.342
C02626=1119.962,29.514,-52.496,179.778,6.906,149.342
C02627=1119.968,29.265,-52.480,179.777,6.902,149.341
C02628=1119.972,29.015,-52.465,179.776,6.897,149.340
C02629=1119.978,28.765,-52.450,179.775,6.893,149.340
C02630=1119.983,28.516,-52.435,179.773,6.889,149.339
C02631=1119.988,28.267,-52.420,179.772,6.884,149.338
C02632=1119.993,28.017,-52.406,179.771,6.880,149.338
C02633=1119.998,27.768,-52.391,179.770,6.876,149.337
C02634=1120.003,27.518,-52.376,179.770,6.871,149.336
C02635=1120.008,27.269,-52.361,179.769,6.867,149.335
C02636=1120.013,27.020,-52.345,179.768,6.862,149.335
C02637=1120.018,26.770,-52.331,179.767,6.858,149.334
C02638=1120.023,26.521,-52.316,179.766,6.854,149.334
C02639=1120.029,26.271,-52.301,179.764,6.850,149.333
C02640=1120.033,26.021,-52.286,179.763,6.845,149.332
C02641=1120.038,25.772,-52.270,179.763,6.841,149.331
C02642=1120.043,25.522,-52.256,179.762,6.836,149.331
C02643=1120.048,25.273,-52.241,179.761,6.833,149.330
C02644=1120.053,25.023,-52.226,179.760,6.828,149.329
C02645=1120.058,24.774,-52.211,179.759,6.824,149.329
C02646=1120.063,24.524,-52.197,179.759,6.819,149.328
C02647=1120.068,24.275,-52.181,179.758,6.815,149.327
C02648=1120.073,24.025,-52.167,179.757,6.811,149.327
C02649=1120.078,23.776,-52.152,179.756,6.806,149.326
C02650=1120.084,23.526,-52.137,179.754,6.802,149.325
C02651=1120.088,23.277,-52.122,179.754,6.797,149.324
C02652=1120.093,23.027,-52.108,179.753,6.793,149.324
C02653=1120.098,22.778,-52.093,179.752,6.789,149.323
C02654=1120.104,22.528,-52.078,179.751,6.784,149.322
C02655=1120.109,22.278,-52.063,179.750,6.780,149.322
C02656=1120.114,22.030,-52.049,179.749,6.775,149.321
C02657=1120.118,21.815,-52.036,179.748,6.771,149.320
C02658=1120.122,21.600,-52.023,179.748,6.768,149.320
C02659=1120.127,21.385,-52.011,179.747,6.764,149.319
C02660=1120.132,21.170,-51.998,179.746,6.760,149.319
C02661=1120.136,20.955,-51.986,179.745,6.757,149.318
C02662=1120.140,20.740,-51.973,179.744,6.752,149.317
C02663=1120.144,20.525,-51.960,179.744,6.749,149.317
C02664=1120.149,20.310,-51.947,179.743,6.744,149.316
C02665=1120.154,20.061,-51.933,179.742,6.740,149.315
C02666=1120.158,19.812,-51.918,179.741,6.735,149.314
C02667=1120.163,19.562,-51.904,179.740,6.731,149.314
C02668=1120.169,19.312,-51.889,179.739,6.727,149.313
C02669=1120.174,19.062,-51.875,179.739,6.722,149.312
C02670=1120.179,18.814,-51.860,179.737,6.718,149.312
C02671=1120.184,18.564,-51.846,179.737,6.713,149.311
C02672=1120.189,18.314,-51.831,179.736,6.709,149.310
C02673=1120.194,18.065,-51.817,179.735,6.704,149.309
C02674=1120.199,17.815,-51.802,179.734,6.700,149.308
C02675=1120.204,17.566,-51.787,179.733,6.695,149.308
C02676=1120.209,17.316,-51.773,179.733,6.691,149.307
C02677=1120.214,17.066,-51.759,179.732,6.686,149.306
C02678=1120.220,16.818,-51.744,179.731,6.682,149.305
C02679=1120.225,16.568,-51.730,179.730,6.677,149.305
C02680=1120.229,16.318,-51.716,179.729,6.673,149.304
C02681=1120.234,16.069,-51.701,179.728,6.668,149.303
C02682=1120.239,15.819,-51.687,179.728,6.664,149.302
C02683=1120.245,15.569,-51.672,179.727,6.659,149.302
C02684=1120.250,15.319,-51.658,179.726,6.654,149.301
C02685=1120.255,15.071,-51.643,179.725,6.650,149.300
C02686=1120.260,14.821,-51.629,179.725,6.645,149.299
C02687=1120.265,14.571,-51.615,179.724,6.641,149.299
C02688=1120.270,14.322,-51.600,179.723,6.636,149.298
C02689=1120.275,14.072,-51.586,179.722,6.632,149.297
C02690=1120.281,13.823,-51.572,179.722,6.627,149.296
C02691=1120.286,13.573,-51.558,179.720,6.623,149.296
C02692=1120.291,13.323,-51.544,179.720,6.618,149.295
C02693=1120.296,13.074,-51.529,179.719,6.614,149.294
C02694=1120.300,12.824,-51.515,179.718,6.609,149.293
C02695=1120.306,12.575,-51.501,179.718,6.605,149.292
C02696=1120.311,12.325,-51.487,179.717,6.600,149.292
C02697=1120.316,12.076,-51.473,179.716,6.596,149.291
C02698=1120.321,11.826,-51.458,179.716,6.591,149.290
C02699=1120.326,11.576,-51.444,179.715,6.587,149.289
C02700=1120.331,11.327,-51.430,179.714,6.582,149.288
C02701=1120.336,11.078,-51.416,179.713,6.577,149.288
C02702=1120.341,10.828,-51.402,179.712,6.573,149.287
C02703=1120.346,10.578,-51.387,179.712,6.568,149.286
C02704=1120.352,10.329,-51.373,179.711,6.563,149.285
C02705=1120.357,10.079,-51.359,179.710,6.559,149.284
C02706=1120.362,9.830,-51.345,179.709,6.554,149.283
C02707=1120.367,9.581,-51.332,179.709,6.549,149.283
C02708=1120.371,9.331,-51.317,179.708,6.544,149.282
C02709=1120.376,9.082,-51.303,179.707,6.540,149.281
C02710=1120.382,8.831,-51.289,179.707,6.535,149.280
C02711=1120.387,8.582,-51.276,179.706,6.530,149.279
C02712=1120.392,8.332,-51.261,179.705,6.526,149.279
C02713=1120.396,8.118,-51.249,179.705,6.522,149.278
C02714=1120.400,7.903,-51.237,179.705,6.519,149.277
C02715=1120.406,7.688,-51.225,179.704,6.514,149.276
C02716=1120.410,7.473,-51.213,179.704,6.510,149.276
C02717=1120.414,7.258,-51.201,179.703,6.507,149.275
C02718=1120.418,7.043,-51.189,179.702,6.502,149.274
C02719=1120.423,6.828,-51.177,179.702,6.499,149.273
C02720=1120.427,6.613,-51.165,179.702,6.495,149.273
C02721=1120.432,6.363,-51.151,179.701,6.490,149.272
C02722=1120.438,6.114,-51.137,179.701,6.486,149.271
C02723=1120.442,5.865,-51.123,179.700,6.481,149.270
C02724=1120.447,5.615,-51.110,179.700,6.476,149.269
C02725=1120.453,5.366,-51.096,179.699,6.473,149.269
C02726=1120.458,5.116,-51.082,179.699,6.468,149.268
C02727=1120.463,4.866,-51.067,179.698,6.463,149.267
C02728=1120.468,4.617,-51.055,179.698,6.458,149.266
C02729=1120.473,4.367,-51.040,179.697,6.454,149.265
C02730=1120.478,4.117,-51.026,179.697,6.449,149.264
C02731=1120.484,3.868,-51.013,179.696,6.445,149.263
C02732=1120.488,3.618,-50.999,179.696,6.441,149.263
C02733=1120.493,3.369,-50.985,179.695,6.436,149.262
C02734=1120.499,3.119,-50.972,179.695,6.431,149.261
C02735=1120.504,2.869,-50.958,179.694,6.427,149.260
C02736=1120.508,2.621,-50.944,179.693,6.422,149.259
C02737=1120.514,2.370,-50.931,179.693,6.418,149.258
C02738=1120.519,2.121,-50.917,179.693,6.414,149.257
C02739=1120.524,1.872,-50.903,179.692,6.409,149.257
C02740=1120.529,1.622,-50.890,179.691,6.405,149.256
C02741=1120.534,1.373,-50.876,179.691,6.400,149.255
C02742=1120.540,1.122,-50.862,179.690,6.395,149.254
C02743=1120.544,0.874,-50.849,179.690,6.390,149.253
C02744=1120.550,0.623,-50.835,179.689,6.386,149.253
C02745=1120.555,0.373,-50.821,179.689,6.382,149.252
C02746=1120.559,0.125,-50.808,179.688,6.377,149.251
C02747=1120.565,-0.126,-50.794,179.688,6.373,149.250
C02748=1120.570,-0.375,-50.780,179.687,6.368,149.249
C02749=1120.575,-0.625,-50.767,179.686,6.364,149.248
C02750=1120.580,-0.874,-50.753,179.685,6.359,149.248
C02751=1120.586,-1.124,-50.740,179.685,6.354,149.247
C02752=1120.590,-1.373,-50.726,179.685,6.351,149.246
C02753=1120.596,-1.623,-50.713,179.684,6.346,149.245
C02754=1120.601,-1.872,-50.699,179.684,6.341,149.244
C02755=1120.606,-2.122,-50.686,179.683,6.336,149.243
C02756=1120.611,-2.371,-50.672,179.682,6.332,149.243
C02757=1120.616,-2.621,-50.659,179.681,6.327,149.242
C02758=1120.622,-2.871,-50.646,179.681,6.323,149.241
C02759=1120.626,-3.120,-50.632,179.680,6.318,149.240
C02760=1120.632,-3.370,-50.619,179.679,6.314,149.239
C02761=1120.637,-3.619,-50.605,179.680,6.310,149.238
C02762=1120.642,-3.869,-50.592,179.679,6.305,149.238
C02763=1120.647,-4.118,-50.578,179.678,6.301,149.237
C02764=1120.652,-4.368,-50.565,179.677,6.296,149.236
C02765=1120.657,-4.618,-50.552,179.677,6.291,149.235
C02766=1120.662,-4.867,-50.538,179.676,6.287,149.234
C02767=1120.667,-5.117,-50.525,179.675,6.282,149.234
C02768=1120.672,-5.366,-50.512,179.675,6.277,149.233
C02769=1120.677,-5.582,-50.500,179.675,6.274,149.232
C02770=1120.681,-5.796,-50.489,179.674,6.270,149.231
C02771=1120.686,-6.011,-50.477,179.673,6.266,149.231
C02772=1120.690,-6.227,-50.466,179.673,6.262,149.230
C02773=1120.694,-6.441,-50.454,179.672,6.258,149.229
C02774=1120.699,-6.657,-50.443,179.672,6.254,149.228
C02775=1120.703,-6.871,-50.431,179.671,6.251,149.228
C02776=1120.708,-7.086,-50.420,179.670,6.246,149.227
C02777=1120.713,-7.336,-50.407,179.670,6.242,149.226
C02778=1120.718,-7.586,-50.394,179.669,6.237,149.226
C02779=1120.723,-7.835,-50.381,179.668,6.233,149.225
C02780=1120.728,-8.085,-50.367,179.669,6.229,149.224
C02781=1120.733,-8.334,-50.354,179.668,6.224,149.223
C02782=1120.739,-8.584,-50.341,179.667,6.220,149.222
C02783=1120.744,-8.834,-50.328,179.667,6.215,149.221
C02784=1120.749,-9.083,-50.314,179.666,6.210,149.221
C02785=1120.754,-9.333,-50.301,179.665,6.206,149.220
C02786=1120.759,-9.582,-50.289,179.665,6.201,149.219
C02787=1120.765,-9.832,-50.275,179.664,6.196,149.218
C02788=1120.769,-10.082,-50.262,179.663,6.192,149.217
C02789=1120.775,-10.332,-50.249,179.663,6.187,149.217
C02790=1120.779,-10.581,-50.235,179.662,6.182,149.216
C02791=1120.784,-10.830,-50.223,179.661,6.178,149.215
C02792=1120.790,-11.080,-50.210,179.661,6.173,149.214
C02793=1120.795,-11.330,-50.197,179.660,6.169,149.213
C02794=1120.800,-11.579,-50.184,179.659,6.164,149.213
C02795=1120.806,-11.829,-50.171,179.659,6.160,149.212
C02796=1120.810,-12.079,-50.158,179.658,6.155,149.211
C02797=1120.815,-12.328,-50.145,179.657,6.151,149.210
C02798=1120.821,-12.578,-50.132,179.657,6.146,149.209
C02799=1120.826,-12.828,-50.119,179.656,6.141,149.208
C02800=1120.831,-13.077,-50.107,179.656,6.136,149.207
C02801=1120.837,-13.327,-50.093,179.655,6.132,149.207
C02802=1120.841,-13.576,-50.080,179.654,6.127,149.206
C02803=1120.846,-13.826,-50.067,179.654,6.123,149.205
C02804=1120.852,-14.075,-50.054,179.653,6.118,149.204
C02805=1120.856,-14.325,-50.041,179.652,6.113,149.203
C02806=1120.862,-14.575,-50.028,179.652,6.109,149.203
C02807=1120.867,-14.824,-50.016,179.651,6.104,149.202
C02808=1120.873,-15.074,-50.003,179.650,6.100,149.201
C02809=1120.877,-15.324,-49.990,179.650,6.095,149.200
C02810=1120.883,-15.573,-49.978,179.649,6.090,149.199
C02811=1120.888,-15.823,-49.965,179.648,6.086,149.199
C02812=1120.893,-16.073,-49.952,179.648,6.081,149.198
C02813=1120.898,-16.322,-49.939,179.647,6.076,149.197
C02814=1120.903,-16.572,-49.926,179.647,6.072,149.196
C02815=1120.908,-16.821,-49.914,179.646,6.067,149.195
C02816=1120.913,-17.071,-49.901,179.645,6.062,149.194
C02817=1120.919,-17.321,-49.888,179.644,6.057,149.193
C02818=1120.924,-17.570,-49.875,179.644,6.052,149.192
C02819=1120.929,-17.819,-49.862,179.643,6.048,149.192
C02820=1120.934,-18.069,-49.850,179.642,6.043,149.191
C02821=1120.939,-18.319,-49.838,179.642,6.039,149.190
C02822=1120.944,-18.569,-49.825,179.641,6.034,149.189
C02823=1120.950,-18.818,-49.812,179.641,6.029,149.188
C02824=1120.955,-19.068,-49.799,179.640,6.025,149.188
C02825=1120.959,-19.283,-49.789,179.639,6.020,149.187
C02826=1120.963,-19.498,-49.777,179.639,6.016,149.186
C02827=1120.968,-19.714,-49.766,179.638,6.012,149.185
C02828=1120.972,-19.928,-49.756,179.638,6.009,149.185
C02829=1120.977,-20.143,-49.745,179.637,6.004,149.184
C02830=1120.982,-20.359,-49.734,179.636,5.999,149.183
C02831=1120.986,-20.573,-49.723,179.636,5.996,149.182
C02832=1120.990,-20.789,-49.712,179.635,5.991,149.182
C02833=1120.995,-21.038,-49.700,179.634,5.987,149.181
C02834=1121.001,-21.288,-49.688,179.634,5.982,149.180
C02835=1121.006,-21.538,-49.675,179.633,5.977,149.179
C02836=1121.011,-21.787,-49.663,179.633,5.973,149.178
C02837=1121.016,-22.036,-49.650,179.632,5.968,149.177
C02838=1121.022,-22.286,-49.638,179.631,5.962,149.176
C02839=1121.027,-22.536,-49.625,179.630,5.958,149.176
C02840=1121.032,-22.786,-49.612,179.630,5.953,149.175
C02841=1121.037,-23.036,-49.600,179.629,5.949,149.174
C02842=1121.042,-23.285,-49.588,179.629,5.944,149.173
C02843=1121.048,-23.535,-49.576,179.628,5.938,149.172
C02844=1121.053,-23.784,-49.563,179.627,5.934,149.171
C02845=1121.058,-24.034,-49.551,179.627,5.929,149.170
C02846=1121.063,-24.284,-49.539,179.626,5.924,149.169
C02847=1121.068,-24.534,-49.526,179.625,5.920,149.169
C02848=1121.073,-24.784,-49.514,179.624,5.914,149.168
C02849=1121.079,-25.033,-49.501,179.624,5.909,149.167
C02850=1121.084,-25.282,-49.489,179.623,5.905,149.166
C02851=1121.089,-25.532,-49.477,179.623,5.900,149.165
C02852=1121.094,-25.781,-49.464,179.622,5.894,149.164
C02853=1121.100,-26.031,-49.452,179.622,5.890,149.163
C02854=1121.105,-26.281,-49.440,179.623,5.886,149.162
C02855=1121.109,-26.530,-49.428,179.623,5.882,149.161
C02856=1121.115,-26.780,-49.416,179.624,5.878,149.160
C02857=1121.120,-27.030,-49.404,179.625,5.874,149.159
C02858=1121.125,-27.279,-49.391,179.626,5.870,149.158
C02859=1121.131,-27.529,-49.379,179.626,5.865,149.157
C02860=1121.135,-27.779,-49.366,179.626,5.861,149.156
C02861=1121.140,-28.029,-49.355,179.627,5.857,149.155
C02862=1121.146,-28.278,-49.342,179.628,5.853,149.153
C02863=1121.151,-28.528,-49.330,179.628,5.849,149.153
C02864=1121.156,-28.777,-49.317,179.628,5.844,149.151
C02865=1121.162,-29.027,-49.306,179.629,5.841,149.151
C02866=1121.167,-29.277,-49.293,179.629,5.836,149.149
C02867=1121.171,-29.526,-49.282,179.629,5.832,149.149
C02868=1121.177,-29.776,-49.269,179.629,5.828,149.148
C02869=1121.182,-30.025,-49.257,179.630,5.824,149.146
C02870=1121.187,-30.275,-49.245,179.630,5.820,149.146
C02871=1121.193,-30.525,-49.233,179.630,5.815,149.145
C02872=1121.198,-30.775,-49.221,179.630,5.811,149.144
C02873=1121.203,-31.024,-49.208,179.630,5.807,149.143
C02874=1121.209,-31.274,-49.196,179.630,5.802,149.142
C02875=1121.213,-31.524,-49.185,179.630,5.798,149.141
C02876=1121.218,-31.773,-49.172,179.630,5.794,149.140
C02877=1121.224,-32.023,-49.161,179.630,5.790,149.139
C02878=1121.229,-32.272,-49.148,179.630,5.786,149.138
C02879=1121.234,-32.522,-49.136,179.630,5.781,149.137
C02880=1121.240,-32.772,-49.124,179.629,5.776,149.136
C02881=1121.244,-32.987,-49.114,179.629,5.773,149.136
C02882=1121.248,-33.202,-49.104,179.628,5.769,149.135
C02883=1121.253,-33.418,-49.093,179.629,5.765,149.134
C02884=1121.257,-33.632,-49.083,179.628,5.762,149.133
C02885=1121.262,-33.848,-49.073,179.627,5.757,149.133
C02886=1121.266,-34.063,-49.062,179.627,5.753,149.132
C02887=1121.270,-34.278,-49.052,179.627,5.750,149.131
C02888=1121.275,-34.493,-49.042,179.627,5.746,149.130
C02889=1121.281,-34.743,-49.029,179.626,5.741,149.130
C02890=1121.285,-34.992,-49.018,179.626,5.737,149.129
C02891=1121.291,-35.242,-49.006,179.625,5.732,149.128
C02892=1121.296,-35.492,-48.994,179.624,5.728,149.127
C02893=1121.301,-35.741,-48.981,179.624,5.723,149.126
C02894=1121.306,-35.991,-48.970,179.622,5.718,149.125
C02895=1121.311,-36.241,-48.958,179.622,5.713,149.125
C02896=1121.317,-36.491,-48.946,179.621,5.709,149.124
C02897=1121.322,-36.740,-48.934,179.621,5.704,149.123
C02898=1121.327,-36.990,-48.922,179.620,5.699,149.122
C02899=1121.333,-37.239,-48.911,179.619,5.694,149.121
C02900=1121.338,-37.489,-48.899,179.618,5.689,149.121
C02901=1121.343,-37.739,-48.888,179.617,5.684,149.120
C02902=1121.348,-37.989,-48.876,179.616,5.679,149.119
C02903=1121.353,-38.238,-48.863,179.615,5.674,149.118
C02904=1121.358,-38.488,-48.852,179.614,5.669,149.117
C02905=1121.363,-38.737,-48.840,179.613,5.664,149.117
C02906=1121.369,-38.987,-48.828,179.612,5.660,149.116
C02907=1121.374,-39.237,-48.817,179.611,5.654,149.115
C02908=1121.380,-39.486,-48.805,179.610,5.649,149.114
C02909=1121.385,-39.736,-48.793,179.608,5.644,149.114
C02910=1121.390,-39.986,-48.782,179.607,5.638,149.113
C02911=1121.395,-40.236,-48.770,179.606,5.634,149.112
C02912=1121.401,-40.486,-48.758,179.605,5.628,149.111
C02913=1121.405,-40.735,-48.747,179.604,5.623,149.110
C02914=1121.411,-40.985,-48.736,179.602,5.618,149.110
C02915=1121.416,-41.234,-48.724,179.601,5.612,149.109
C02916=1121.421,-41.484,-48.712,179.599,5.606,149.108
C02917=1121.427,-41.734,-48.701,179.598,5.601,149.107
C02918=1121.432,-41.984,-48.689,179.596,5.596,149.107
C02919=1121.438,-42.233,-48.678,179.595,5.590,149.106
C02920=1121.442,-42.483,-48.666,179.593,5.584,149.105
C02921=1121.448,-42.732,-48.655,179.592,5.579,149.104
C02922=1121.452,-42.982,-48.643,179.590,5.573,149.104
C02923=1121.458,-43.231,-48.632,179.590,5.568,149.103
C02924=1121.463,-43.481,-48.620,179.590,5.564,149.101
C02925=1121.469,-43.731,-48.609,179.590,5.558,149.100
C02926=1121.474,-43.981,-48.598,179.591,5.554,149.099
C02927=1121.479,-44.231,-48.586,179.591,5.549,149.098
C02928=1121.484,-44.480,-48.575,179.591,5.544,149.097
C02929=1121.489,-44.730,-48.564,179.591,5.540,149.096
C02930=1121.494,-44.980,-48.552,179.591,5.535,149.095
C02931=1121.500,-45.228,-48.541,179.591,5.531,149.094
C02932=1121.505,-45.479,-48.530,179.592,5.526,149.093
C02933=1121.510,-45.729,-48.519,179.592,5.521,149.092
C02934=1121.516,-45.979,-48.507,179.592,5.516,149.091
C02935=1121.521,-46.228,-48.496,179.592,5.511,149.090
C02936=1121.526,-46.477,-48.484,179.593,5.507,149.088
C02937=1121.531,-46.693,-48.475,179.593,5.503,149.088
C02938=1121.535,-46.908,-48.465,179.592,5.498,149.087
C02939=1121.540,-47.123,-48.455,179.592,5.494,149.086
C02940=1121.544,-47.338,-48.445,179.593,5.490,149.085
C02941=1121.549,-47.554,-48.436,179.593,5.487,149.084
C02942=1121.553,-47.769,-48.426,179.593,5.483,149.083
C02943=1121.557,-47.985,-48.416,179.593,5.479,149.082
C02944=1121.562,-48.200,-48.407,179.594,5.474,149.081
C02945=1121.568,-48.449,-48.396,179.593,5.470,149.080
C02946=1121.573,-48.699,-48.384,179.594,5.465,149.079
C02947=1121.577,-48.949,-48.373,179.594,5.460,149.078
C02948=1121.584,-49.199,-48.362,179.594,5.456,149.077
C02949=1121.588,-49.448,-48.351,179.594,5.451,149.076
C02950=1121.594,-49.698,-48.339,179.594,5.446,149.075
C02951=1121.599,-49.948,-48.329,179.595,5.442,149.074
C02952=1121.604,-50.197,-48.318,179.595,5.437,149.072
C02953=1121.610,-50.447,-48.306,179.595,5.432,149.071
C02954=1121.615,-50.697,-48.295,179.595,5.427,149.070
C02955=1121.620,-50.946,-48.284,179.595,5.423,149.069
C02956=1121.625,-51.196,-48.272,179.596,5.418,149.068
C02957=1121.631,-51.446,-48.262,179.596,5.413,149.067
C02958=1121.636,-51.695,-48.251,179.596,5.409,149.066
C02959=1121.641,-51.945,-48.239,179.596,5.404,149.065
C02960=1121.647,-52.195,-48.229,179.596,5.399,149.064
C02961=1121.651,-52.445,-48.217,179.596,5.395,149.063
C02962=1121.657,-52.694,-48.207,179.596,5.390,149.062
C02963=1121.662,-52.944,-48.195,179.597,5.385,149.061
C02964=1121.667,-53.194,-48.184,179.597,5.381,149.060
C02965=1121.673,-53.443,-48.174,179.597,5.376,149.058
C02966=1121.678,-53.693,-48.162,179.597,5.371,149.057
C02967=1121.683,-53.943,-48.151,179.598,5.366,149.056
C02968=1121.688,-54.192,-48.140,179.598,5.362,149.055
C02969=1121.693,-54.442,-48.129,179.598,5.357,149.054
C02970=1121.699,-54.692,-48.118,179.599,5.353,149.053
C02971=1121.704,-54.941,-48.107,179.598,5.348,149.052
C02972=1121.709,-55.192,-48.096,179.599,5.343,149.051
C02973=1121.714,-55.441,-48.086,179.599,5.338,149.050
C02974=1121.720,-55.691,-48.074,179.599,5.334,149.049
C02975=1121.725,-55.940,-48.063,179.599,5.329,149.048
C02976=1121.730,-56.190,-48.053,179.599,5.324,149.047
C02977=1121.735,-56.440,-48.042,179.599,5.320,149.046
C02978=1121.741,-56.690,-48.031,179.600,5.315,149.044
C02979=1121.746,-56.939,-48.019,179.600,5.311,149.044
C02980=1121.752,-57.189,-48.009,179.600,5.306,149.042
C02981=1121.756,-57.439,-47.998,179.600,5.301,149.041
C02982=1121.762,-57.688,-47.988,179.600,5.297,149.040
C02983=1121.767,-57.938,-47.976,179.600,5.292,149.039
C02984=1121.772,-58.188,-47.966,179.601,5.287,149.038
C02985=1121.778,-58.438,-47.955,179.601,5.283,149.037
C02986=1121.783,-58.688,-47.944,179.601,5.278,149.036
C02987=1121.788,-58.937,-47.934,179.601,5.273,149.035
C02988=1121.793,-59.187,-47.922,179.601,5.268,149.034
C02989=1121.799,-59.436,-47.912,179.602,5.264,149.033
C02990=1121.803,-59.686,-47.901,179.601,5.259,149.032
C02991=1121.809,-59.935,-47.891,179.602,5.255,149.031
C02992=1121.815,-60.186,-47.879,179.602,5.250,149.029
C02993=1121.818,-60.401,-47.871,179.601,5.245,149.029
C02994=1121.823,-60.617,-47.861,179.600,5.241,149.028
C02995=1121.827,-60.832,-47.851,179.600,5.236,149.027
C02996=1121.832,-61.047,-47.842,179.599,5.232,149.027
C02997=1121.837,-61.262,-47.833,179.599,5.227,149.026
C02998=1121.842,-61.477,-47.824,179.598,5.223,149.025
C02999=1121.846,-61.692,-47.815,179.597,5.218,149.024
C03000=1121.851,-61.908,-47.806,179.596,5.214,149.023
C03001=1121.856,-62.158,-47.795,179.596,5.209,149.022
C03002=1121.861,-62.408,-47.785,179.595,5.203,149.021
C03003=1121.866,-62.657,-47.774,179.595,5.198,149.021
C03004=1121.872,-62.907,-47.763,179.594,5.193,149.020
C03005=1121.877,-63.157,-47.753,179.593,5.187,149.019
C03006=1121.883,-63.407,-47.742,179.592,5.183,149.018
C03007=1121.887,-63.657,-47.731,179.592,5.177,149.017
C03008=1121.893,-63.906,-47.721,179.591,5.172,149.016
C03009=1121.899,-64.156,-47.711,179.590,5.166,149.015
C03010=1121.904,-64.406,-47.700,179.590,5.162,149.014
C03011=1121.909,-64.655,-47.689,179.589,5.156,149.013
C03012=1121.914,-64.905,-47.679,179.589,5.151,149.012
C03013=1121.920,-65.155,-47.668,179.588,5.145,149.011
C03014=1121.925,-65.405,-47.658,179.588,5.141,149.010
C03015=1121.930,-65.654,-47.648,179.587,5.135,149.009
C03016=1121.935,-65.904,-47.638,179.587,5.130,149.008
C03017=1121.940,-66.154,-47.627,179.586,5.124,149.007
C03018=1121.945,-66.403,-47.616,179.586,5.119,149.006
C03019=1121.950,-66.653,-47.606,179.585,5.114,149.005
C03020=1121.956,-66.903,-47.596,179.585,5.109,149.004
C03021=1121.961,-67.152,-47.585,179.584,5.103,149.003
C03022=1121.966,-67.402,-47.575,179.584,5.098,149.002
C03023=1121.972,-67.652,-47.565,179.584,5.093,149.001
C03024=1121.978,-67.902,-47.554,179.583,5.087,149.000
C03025=1121.983,-68.152,-47.544,179.583,5.083,148.999
C03026=1121.988,-68.401,-47.534,179.582,5.077,148.998
C03027=1121.994,-68.651,-47.523,179.582,5.072,148.997
C03028=1121.998,-68.901,-47.513,179.581,5.066,148.996
C03029=1122.004,-69.150,-47.503,179.581,5.061,148.995
C03030=1122.009,-69.400,-47.493,179.581,5.056,148.994
C03031=1122.014,-69.650,-47.482,179.580,5.050,148.993
C03032=1122.020,-69.900,-47.472,179.580,5.045,148.992
C03033=1122.026,-70.149,-47.462,179.580,5.040,148.991
C03034=1122.031,-70.399,-47.451,179.580,5.035,148.989
C03035=1122.035,-70.649,-47.442,179.579,5.030,148.989
C03036=1122.041,-70.898,-47.432,179.579,5.025,148.987
C03037=1122.046,-71.148,-47.421,179.579,5.019,148.986
C03038=1122.052,-71.398,-47.411,179.579,5.014,148.985
C03039=1122.057,-71.648,-47.401,179.579,5.009,148.984
C03040=1122.062,-71.897,-47.392,179.578,5.003,148.983
C03041=1122.067,-72.148,-47.381,179.578,4.998,148.982
C03042=1122.073,-72.397,-47.371,179.578,4.993,148.981
C03043=1122.079,-72.647,-47.361,179.578,4.987,148.980
C03044=1122.084,-72.896,-47.351,179.577,4.982,148.979
C03045=1122.088,-73.146,-47.341,179.577,4.977,148.978
C03046=1122.094,-73.396,-47.330,179.577,4.972,148.977
C03047=1122.100,-73.646,-47.321,179.577,4.966,148.975
C03048=1122.105,-73.895,-47.311,179.577,4.961,148.974
C03049=1122.109,-74.111,-47.302,179.576,4.956,148.973
C03050=1122.114,-74.327,-47.293,179.577,4.952,148.972
C03051=1122.118,-74.542,-47.285,179.577,4.947,148.971
C03052=1122.124,-74.757,-47.277,179.577,4.943,148.970
C03053=1122.128,-74.973,-47.268,179.577,4.938,148.970
C03054=1122.132,-75.188,-47.259,179.576,4.934,148.969
C03055=1122.137,-75.404,-47.251,179.576,4.930,148.968
C03056=1122.142,-75.619,-47.242,179.576,4.925,148.967
C03057=1122.148,-75.869,-47.232,179.576,4.920,148.966
C03058=1122.152,-76.119,-47.222,179.576,4.915,148.964
C03059=1122.158,-76.368,-47.212,179.577,4.909,148.963
C03060=1122.163,-76.618,-47.202,179.577,4.904,148.962
C03061=1122.168,-76.868,-47.193,179.576,4.898,148.961
C03062=1122.174,-77.117,-47.183,179.576,4.893,148.960
C03063=1122.179,-77.367,-47.172,179.577,4.888,148.959
C03064=1122.184,-77.617,-47.163,179.577,4.883,148.957
C03065=1122.190,-77.867,-47.153,179.576,4.878,148.957
C03066=1122.195,-78.116,-47.143,179.577,4.873,148.955
C03067=1122.200,-78.366,-47.134,179.577,4.868,148.954
C03068=1122.206,-78.616,-47.124,179.577,4.863,148.953
C03069=1122.211,-78.865,-47.114,179.577,4.858,148.952
C03070=1122.216,-79.116,-47.104,179.577,4.852,148.951
C03071=1122.222,-79.365,-47.094,179.577,4.847,148.949
C03072=1122.227,-79.615,-47.085,179.577,4.842,148.948
C03073=1122.233,-79.865,-47.075,179.578,4.837,148.947
C03074=1122.237,-80.114,-47.065,179.578,4.832,148.946
C03075=1122.243,-80.364,-47.056,179.578,4.827,148.945
C03076=1122.249,-80.614,-47.046,179.578,4.821,148.944
C03077=1122.254,-80.864,-47.036,179.578,4.816,148.942
C03078=1122.259,-81.114,-47.026,179.578,4.811,148.941
C03079=1122.264,-81.364,-47.017,179.579,4.806,148.940
C03080=1122.270,-81.613,-47.007,179.579,4.801,148.939
C03081=1122.275,-81.862,-46.997,179.579,4.796,148.938
C03082=1122.281,-82.113,-46.988,179.580,4.790,148.936
C03083=1122.286,-82.362,-46.978,179.580,4.785,148.935
C03084=1122.291,-82.612,-46.969,179.580,4.780,148.934
C03085=1122.296,-82.861,-46.959,179.580,4.775,148.933
C03086=1122.302,-83.111,-46.950,179.581,4.770,148.932
C03087=1122.307,-83.361,-46.940,179.581,4.765,148.931
C03088=1122.312,-83.612,-46.930,179.581,4.760,148.929
C03089=1122.317,-83.861,-46.921,179.581,4.755,148.928
C03090=1122.323,-84.111,-46.911,179.582,4.750,148.927
C03091=1122.328,-84.360,-46.901,179.582,4.744,148.926
C03092=1122.334,-84.610,-46.892,179.583,4.740,148.924
C03093=1122.339,-84.860,-46.883,179.583,4.735,148.923
C03094=1122.345,-85.110,-46.873,179.583,4.729,148.922
C03095=1122.350,-85.360,-46.864,179.584,4.724,148.921
C03096=1122.355,-85.609,-46.854,179.584,4.719,148.920
C03097=1122.361,-85.859,-46.845,179.584,4.715,148.919
C03098=1122.366,-86.108,-46.835,179.585,4.710,148.917
C03099=1122.371,-86.358,-46.826,179.585,4.704,148.916
C03100=1122.376,-86.608,-46.817,179.586,4.699,148.915
C03101=1122.382,-86.858,-46.807,179.586,4.694,148.914
C03102=1122.387,-87.108,-46.798,179.586,4.689,148.912
C03103=1122.393,-87.357,-46.788,179.587,4.684,148.911
C03104=1122.398,-87.607,-46.779,179.587,4.680,148.910
C03105=1122.402,-87.823,-46.771,179.588,4.675,148.909
C03106=1122.407,-88.039,-46.762,179.588,4.671,148.908
C03107=1122.412,-88.254,-46.754,179.589,4.666,148.907
C03108=1122.416,-88.470,-46.746,179.589,4.662,148.906
C03109=1122.421,-88.685,-46.738,179.590,4.658,148.905
C03110=1122.426,-88.900,-46.730,179.590,4.654,148.904
C03111=1122.430,-89.116,-46.722,179.591,4.650,148.903
C03112=1122.435,-89.331,-46.714,179.591,4.646,148.902
C03113=1122.441,-89.581,-46.704,179.592,4.640,148.900
C03114=1122.445,-89.831,-46.695,179.593,4.636,148.899
C03115=1122.451,-90.081,-46.686,179.593,4.631,148.898
C03116=1122.457,-90.331,-46.676,179.593,4.626,148.897
C03117=1122.462,-90.581,-46.668,179.594,4.621,148.895
C03118=1122.467,-90.830,-46.658,179.595,4.616,148.894
C03119=1122.472,-91.080,-46.648,179.595,4.611,148.893
C03120=1122.478,-91.330,-46.640,179.596,4.607,148.892
C03121=1122.483,-91.580,-46.631,179.596,4.602,148.890
C03122=1122.488,-91.829,-46.620,179.597,4.597,148.889
C03123=1122.494,-92.079,-46.612,179.598,4.592,148.888
C03124=1122.499,-92.329,-46.603,179.598,4.587,148.887
C03125=1122.505,-92.579,-46.593,179.599,4.582,148.885
C03126=1122.510,-92.828,-46.584,179.599,4.578,148.884
C03127=1122.515,-93.078,-46.575,179.601,4.573,148.883
C03128=1122.521,-93.328,-46.565,179.601,4.568,148.882
C03129=1122.526,-93.578,-46.556,179.602,4.564,148.880
C03130=1122.531,-93.827,-46.547,179.602,4.559,148.879
C03131=1122.537,-94.077,-46.538,179.603,4.554,148.878
C03132=1122.542,-94.327,-46.529,179.604,4.549,148.877
C03133=1122.547,-94.577,-46.520,179.604,4.544,148.876
C03134=1122.553,-94.826,-46.511,179.605,4.540,148.874
C03135=1122.559,-95.077,-46.501,179.605,4.535,148.873
C03136=1122.563,-95.326,-46.492,179.605,4.530,148.872
C03137=1122.569,-95.576,-46.483,179.606,4.524,148.871
C03138=1122.574,-95.825,-46.474,179.606,4.520,148.870
C03139=1122.580,-96.076,-46.464,179.606,4.515,148.869
C03140=1122.585,-96.325,-46.456,179.606,4.510,148.867
C03141=1122.590,-96.575,-46.447,179.607,4.505,148.866
C03142=1122.595,-96.825,-46.438,179.607,4.501,148.865
C03143=1122.602,-97.075,-46.429,179.608,4.495,148.864
C03144=1122.606,-97.324,-46.419,179.608,4.490,148.863
C03145=1122.612,-97.574,-46.410,179.608,4.485,148.862
C03146=1122.617,-97.824,-46.401,179.608,4.480,148.860
C03147=1122.623,-98.074,-46.392,179.609,4.476,148.859
C03148=1122.628,-98.324,-46.383,179.609,4.470,148.858
C03149=1122.633,-98.573,-46.374,179.609,4.465,148.857
C03150=1122.639,-98.823,-46.365,179.610,4.460,148.856
C03151=1122.644,-99.072,-46.356,179.610,4.455,148.854
C03152=1122.650,-99.323,-46.347,179.610,4.451,148.853
C03153=1122.655,-99.572,-46.338,179.610,4.446,148.852
C03154=1122.660,-99.822,-46.329,179.611,4.441,148.851
C03155=1122.665,-100.072,-46.320,179.611,4.435,148.850
C03156=1122.671,-100.322,-46.311,179.611,4.430,148.849
C03157=1122.676,-100.571,-46.303,179.611,4.425,148.847
C03158=1122.682,-100.821,-46.293,179.612,4.421,148.846
C03159=1122.687,-101.071,-46.284,179.612,4.416,148.845
C03160=1122.693,-101.321,-46.276,179.612,4.410,148.844
C03161=1122.697,-101.536,-46.268,179.613,4.406,148.843
C03162=1122.702,-101.752,-46.260,179.612,4.402,148.842
C03163=1122.707,-101.968,-46.253,179.613,4.398,148.841
C03164=1122.711,-102.183,-46.245,179.614,4.393,148.840
C03165=1122.716,-102.399,-46.238,179.613,4.389,148.839
C03166=1122.720,-102.614,-46.230,179.614,4.385,148.838
C03167=1122.725,-102.830,-46.223,179.614,4.381,148.837
C03168=1122.729,-103.046,-46.215,179.614,4.375,148.836
C03169=1122.734,-103.296,-46.206,179.614,4.370,148.835
C03170=1122.740,-103.545,-46.197,179.615,4.365,148.833
C03171=1122.745,-103.795,-46.188,179.615,4.361,148.832
C03172=1122.751,-104.045,-46.179,179.615,4.356,148.831
C03173=1122.756,-104.295,-46.170,179.615,4.351,148.830
C03174=1122.762,-104.545,-46.162,179.616,4.346,148.829
C03175=1122.768,-104.794,-46.153,179.616,4.340,148.828
C03176=1122.773,-105.044,-46.144,179.616,4.335,148.827
C03177=1122.778,-105.294,-46.135,179.616,4.330,148.825
C03178=1122.783,-105.544,-46.127,179.617,4.325,148.824
C03179=1122.789,-105.793,-46.118,179.617,4.320,148.823
C03180=1122.794,-106.043,-46.109,179.617,4.315,148.822
C03181=1122.800,-106.293,-46.101,179.617,4.309,148.821
C03182=1122.805,-106.543,-46.092,179.618,4.305,148.819
C03183=1122.811,-106.792,-46.083,179.618,4.300,148.818
C03184=1122.816,-107.042,-46.075,179.618,4.295,148.817
C03185=1122.821,-107.292,-46.066,179.618,4.290,148.816
C03186=1122.826,-107.543,-46.057,179.619,4.285,148.815
C03187=1122.832,-107.792,-46.049,179.619,4.280,148.814
C03188=1122.837,-108.042,-46.040,179.619,4.274,148.812
C03189=1122.842,-108.291,-46.031,179.619,4.269,148.811
C03190=1122.849,-108.541,-46.023,179.620,4.264,148.810
C03191=1122.854,-108.791,-46.014,179.620,4.259,148.809
C03192=1122.859,-109.041,-46.006,179.620,4.254,148.808
C03193=1122.865,-109.290,-45.997,179.620,4.249,148.806
C03194=1122.869,-109.540,-45.989,179.621,4.243,148.805
C03195=1122.875,-109.790,-45.981,179.621,4.238,148.804
C03196=1122.880,-110.040,-45.972,179.621,4.233,148.803
C03197=1122.886,-110.290,-45.964,179.621,4.228,148.802
C03198=1122.891,-110.540,-45.955,179.622,4.223,148.800
C03199=1122.896,-110.789,-45.946,179.622,4.218,148.799
C03200=1122.902,-111.039,-45.938,179.622,4.212,148.798
C03201=1122.907,-111.289,-45.929,179.622,4.207,148.797
C03202=1122.912,-111.539,-45.920,179.623,4.202,148.796
C03203=1122.919,-111.789,-45.913,179.623,4.197,148.794
C03204=1122.924,-112.038,-45.904,179.623,4.192,148.793
C03205=1122.928,-112.288,-45.895,179.623,4.187,148.792
C03206=1122.934,-112.538,-45.888,179.623,4.182,148.791
C03207=1122.939,-112.788,-45.879,179.623,4.176,148.790
C03208=1122.945,-113.037,-45.871,179.623,4.171,148.789
C03209=1122.951,-113.287,-45.862,179.623,4.165,148.788
C03210=1122.956,-113.537,-45.853,179.624,4.160,148.786
C03211=1122.962,-113.787,-45.845,179.624,4.155,148.785
C03212=1122.966,-114.036,-45.837,179.624,4.150,148.784
C03213=1122.972,-114.287,-45.829,179.624,4.145,148.783
C03214=1122.978,-114.536,-45.820,179.625,4.140,148.781
C03215=1122.983,-114.786,-45.812,179.625,4.134,148.780
C03216=1122.989,-115.036,-45.804,179.625,4.129,148.779
C03217=1122.993,-115.252,-45.796,179.625,4.124,148.778
C03218=1122.997,-115.467,-45.789,179.626,4.120,148.777
C03219=1123.002,-115.683,-45.782,179.625,4.115,148.776
C03220=1123.007,-115.899,-45.775,179.626,4.110,148.775
C03221=1123.012,-116.114,-45.767,179.626,4.106,148.774
C03222=1123.017,-116.330,-45.761,179.626,4.101,148.773
C03223=1123.021,-116.546,-45.754,179.627,4.097,148.772
C03224=1123.026,-116.762,-45.747,179.626,4.092,148.771
C03225=1123.031,-117.012,-45.738,179.627,4.087,148.769
C03226=1123.037,-117.261,-45.730,179.627,4.082,148.768
C03227=1123.042,-117.511,-45.721,179.627,4.077,148.767
C03228=1123.048,-117.761,-45.714,179.627,4.071,148.766
C03229=1123.053,-118.010,-45.705,179.627,4.065,148.765
C03230=1123.059,-118.260,-45.697,179.627,4.060,148.763
C03231=1123.064,-118.511,-45.689,179.628,4.055,148.762
C03232=1123.069,-118.759,-45.681,179.628,4.050,148.761
C03233=1123.075,-119.010,-45.673,179.628,4.045,148.760
C03234=1123.081,-119.259,-45.665,179.628,4.039,148.759
C03235=1123.085,-119.509,-45.657,179.629,4.033,148.757
C03236=1123.091,-119.759,-45.649,179.629,4.028,148.756
C03237=1123.097,-120.009,-45.640,179.629,4.023,148.755
C03238=1123.101,-120.259,-45.633,179.630,4.018,148.754
C03239=1123.107,-120.509,-45.625,179.629,4.012,148.752
C03240=1123.113,-120.759,-45.616,179.630,4.006,148.751
C03241=1123.118,-121.008,-45.609,179.630,4.001,148.750
C03242=1123.123,-121.259,-45.601,179.630,3.996,148.749
C03243=1123.129,-121.508,-45.592,179.630,3.990,148.748
C03244=1123.134,-121.758,-45.584,179.630,3.985,148.746
C03245=1123.140,-122.008,-45.577,179.630,3.980,148.745
C03246=1123.146,-122.257,-45.568,179.631,3.974,148.744
C03247=1123.150,-122.507,-45.561,179.631,3.968,148.742
C03248=1123.156,-122.757,-45.553,179.631,3.963,148.741
C03249=1123.162,-123.007,-45.545,179.632,3.958,148.740
C03250=1123.167,-123.256,-45.537,179.631,3.952,148.739
C03251=1123.172,-123.507,-45.528,179.632,3.947,148.738
C03252=1123.178,-123.756,-45.521,179.632,3.942,148.736
C03253=1123.183,-124.006,-45.513,179.632,3.936,148.735
C03254=1123.188,-124.255,-45.505,179.632,3.930,148.734
C03255=1123.194,-124.506,-45.497,179.633,3.925,148.733
C03256=1123.200,-124.756,-45.489,179.632,3.919,148.731
C03257=1123.205,-125.005,-45.482,179.633,3.914,148.730
C03258=1123.211,-125.255,-45.474,179.633,3.908,148.729
C03259=1123.216,-125.505,-45.466,179.633,3.902,148.728
C03260=1123.221,-125.755,-45.458,179.634,3.897,148.726
C03261=1123.226,-126.004,-45.450,179.634,3.892,148.725
C03262=1123.233,-126.254,-45.443,179.634,3.886,148.724
C03263=1123.237,-126.504,-45.435,179.634,3.881,148.723
C03264=1123.243,-126.754,-45.427,179.634,3.875,148.721
C03265=1123.248,-127.004,-45.420,179.634,3.869,148.720
C03266=1123.254,-127.254,-45.412,179.635,3.864,148.719
C03267=1123.260,-127.503,-45.405,179.634,3.858,148.717
C03268=1123.265,-127.754,-45.396,179.635,3.853,148.716
C03269=1123.270,-128.003,-45.388,179.635,3.847,148.715
C03270=1123.276,-128.252,-45.381,179.635,3.841,148.714
C03271=1123.281,-128.503,-45.373,179.636,3.836,148.712
C03272=1123.287,-128.752,-45.365,179.635,3.830,148.711
C03273=1122.864,-128.743,-45.391,179.643,3.835,148.710
C03274=1122.858,-128.493,-45.399,179.642,3.840,148.711
C03275=1122.853,-128.244,-45.407,179.643,3.846,148.712
C03276=1122.847,-127.993,-45.415,179.642,3.851,148.714
C03277=1122.842,-127.744,-45.422,179.643,3.857,148.715
C03278=1122.837,-127.493,-45.430,179.642,3.862,148.716
C03279=1122.831,-127.244,-45.437,179.641,3.868,148.717
C03280=1122.825,-126.994,-45.445,179.642,3.874,148.719
C03281=1122.820,-126.744,-45.453,179.641,3.879,148.720
C03282=1122.815,-126.495,-45.461,179.641,3.885,148.721
C03283=1122.810,-126.245,-45.469,179.641,3.890,148.723
C03284=1122.804,-125.995,-45.477,179.640,3.896,148.724
C03285=1122.798,-125.745,-45.484,179.641,3.902,148.725
C03286=1122.793,-125.495,-45.492,179.640,3.907,148.726
C03287=1122.787,-125.246,-45.501,179.640,3.912,148.727
C03288=1122.783,-124.996,-45.508,179.640,3.918,148.729
C03289=1122.776,-124.746,-45.516,179.640,3.923,148.730
C03290=1122.772,-124.496,-45.524,179.639,3.929,148.731
C03291=1122.766,-124.246,-45.531,179.640,3.935,148.732
C03292=1122.760,-123.997,-45.540,179.639,3.940,148.734
C03293=1122.755,-123.747,-45.548,179.639,3.945,148.735
C03294=1122.749,-123.497,-45.555,179.639,3.951,148.736
C03295=1122.744,-123.247,-45.563,179.639,3.957,148.738
C03296=1122.739,-122.998,-45.571,179.638,3.962,148.739
C03297=1122.733,-122.747,-45.580,179.638,3.967,148.740
C03298=1122.728,-122.498,-45.587,179.638,3.973,148.741
C03299=1122.723,-122.248,-45.596,179.638,3.978,148.742
C03300=1122.717,-121.998,-45.604,179.638,3.983,148.744
C03301=1122.712,-121.748,-45.611,179.638,3.989,148.745
C03302=1122.706,-121.498,-45.619,179.637,3.995,148.746
C03303=1122.701,-121.248,-45.628,179.637,4.000,148.747
C03304=1122.695,-120.999,-45.635,179.637,4.005,148.749
C03305=1122.690,-120.748,-45.643,179.636,4.010,148.750
C03306=1122.684,-120.499,-45.652,179.637,4.016,148.751
C03307=1122.679,-120.249,-45.659,179.636,4.021,148.752
C03308=1122.673,-120.000,-45.668,179.636,4.027,148.753
C03309=1122.668,-119.749,-45.676,179.636,4.032,148.755
C03310=1122.663,-119.500,-45.683,179.636,4.038,148.756
C03311=1122.657,-119.250,-45.692,179.636,4.043,148.757
C03312=1122.651,-119.000,-45.700,179.635,4.048,148.758
C03313=1122.646,-118.751,-45.709,179.635,4.054,148.760
C03314=1122.642,-118.500,-45.717,179.634,4.059,148.761
C03315=1122.635,-118.251,-45.724,179.635,4.065,148.762
C03316=1122.630,-118.001,-45.733,179.634,4.070,148.763
C03317=1122.624,-117.751,-45.741,179.634,4.075,148.765
C03318=1122.620,-117.501,-45.749,179.634,4.080,148.766
C03319=1122.614,-117.252,-45.757,179.634,4.086,148.767
C03320=1122.609,-117.002,-45.766,179.633,4.091,148.768
C03321=1122.602,-116.752,-45.774,179.633,4.096,148.769
C03322=1122.598,-116.536,-45.782,179.633,4.101,148.770
C03323=1122.594,-116.321,-45.788,179.633,4.106,148.772
C03324=1122.589,-116.105,-45.795,179.633,4.110,148.773
C03325=1122.585,-115.889,-45.803,179.633,4.115,148.773
C03326=1122.579,-115.674,-45.810,179.632,4.119,148.775
C03327=1122.574,-115.458,-45.817,179.632,4.124,148.776
C03328=1122.571,-115.242,-45.824,179.632,4.128,148.777
C03329=1122.566,-115.027,-45.831,179.632,4.133,148.778
C03330=1122.561,-114.777,-45.840,179.631,4.138,148.779
C03331=1122.554,-114.527,-45.848,179.631,4.143,148.780
C03332=1122.549,-114.277,-45.857,179.631,4.148,148.781
C03333=1122.544,-114.027,-45.865,179.631,4.154,148.783
C03334=1122.538,-113.778,-45.873,179.630,4.159,148.784
C03335=1122.534,-113.528,-45.882,179.630,4.164,148.785
C03336=1122.528,-113.278,-45.890,179.630,4.170,148.786
C03337=1122.522,-113.028,-45.898,179.630,4.175,148.787
C03338=1122.517,-112.778,-45.907,179.630,4.180,148.789
C03339=1122.511,-112.529,-45.915,179.630,4.186,148.790
C03340=1122.506,-112.279,-45.924,179.629,4.191,148.791
C03341=1122.500,-112.029,-45.932,179.630,4.195,148.792
C03342=1122.495,-111.779,-45.941,179.629,4.201,148.793
C03343=1122.490,-111.530,-45.950,179.629,4.206,148.794
C03344=1122.485,-111.279,-45.957,179.629,4.211,148.796
C03345=1122.479,-111.030,-45.966,179.629,4.216,148.797
C03346=1122.474,-110.780,-45.975,179.628,4.221,148.798
C03347=1122.468,-110.530,-45.983,179.628,4.226,148.799
C03348=1122.463,-110.281,-45.991,179.628,4.232,148.800
C03349=1122.457,-110.031,-46.000,179.628,4.237,148.802
C03350=1122.452,-109.781,-46.009,179.627,4.242,148.803
C03351=1122.447,-109.531,-46.017,179.627,4.247,148.804
C03352=1122.441,-109.281,-46.026,179.627,4.252,148.805
C03353=1122.436,-109.032,-46.035,179.627,4.258,148.806
C03354=1122.430,-108.781,-46.043,179.626,4.263,148.808
C03355=1122.425,-108.532,-46.052,179.626,4.268,148.809
C03356=1122.420,-108.282,-46.060,179.626,4.273,148.810
C03357=1122.414,-108.032,-46.069,179.626,4.278,148.811
C03358=1122.409,-107.782,-46.078,179.625,4.283,148.812
C03359=1122.403,-107.533,-46.086,179.625,4.289,148.814
C03360=1122.398,-107.283,-46.095,179.625,4.294,148.815
C03361=1122.393,-107.033,-46.104,179.625,4.299,148.816
C03362=1122.388,-106.783,-46.113,179.624,4.304,148.817
C03363=1122.382,-106.534,-46.121,179.625,4.309,148.818
C03364=1122.377,-106.284,-46.130,179.625,4.314,148.819
C03365=1122.371,-106.034,-46.138,179.624,4.318,148.820
C03366=1122.366,-105.784,-46.147,179.623,4.324,148.822
C03367=1122.360,-105.535,-46.156,179.623,4.329,148.823
C03368=1122.355,-105.285,-46.165,179.623,4.334,148.824
C03369=1122.350,-105.035,-46.174,179.623,4.339,148.825
C03370=1122.345,-104.785,-46.183,179.623,4.344,148.826
C03371=1122.340,-104.535,-46.191,179.622,4.349,148.828
C03372=1122.334,-104.285,-46.199,179.622,4.355,148.829
C03373=1122.328,-104.036,-46.208,179.622,4.360,148.830
C03374=1122.323,-103.786,-46.217,179.622,4.365,148.831
C03375=1122.317,-103.536,-46.227,179.621,4.370,148.832
C03376=1122.312,-103.286,-46.235,179.621,4.374,148.834
C03377=1122.306,-103.037,-46.244,179.621,4.379,148.835
C03378=1122.302,-102.821,-46.252,179.621,4.384,148.836
C03379=1122.297,-102.606,-46.260,179.620,4.388,148.837
C03380=1122.293,-102.389,-46.267,179.620,4.392,148.838
C03381=1122.288,-102.174,-46.274,179.620,4.397,148.839
C03382=1122.284,-101.958,-46.282,179.619,4.401,148.840
C03383=1122.279,-101.743,-46.290,179.619,4.405,148.841
C03384=1122.275,-101.527,-46.298,179.619,4.410,148.842
C03385=1122.270,-101.312,-46.305,179.619,4.414,148.843
C03386=1122.264,-101.062,-46.314,179.619,4.419,148.844
C03387=1122.259,-100.812,-46.323,179.619,4.424,148.845
C03388=1122.253,-100.562,-46.332,179.618,4.429,148.846
C03389=1122.248,-100.312,-46.341,179.618,4.434,148.847
C03390=1122.242,-100.063,-46.350,179.617,4.439,148.849
C03391=1122.238,-99.814,-46.359,179.617,4.444,148.850
C03392=1122.232,-99.564,-46.368,179.617,4.450,148.851
C03393=1122.227,-99.314,-46.378,179.617,4.455,148.852
C03394=1122.221,-99.064,-46.387,179.616,4.459,148.853
C03395=1122.216,-98.814,-46.395,179.616,4.464,148.855
C03396=1122.211,-98.564,-46.404,179.616,4.469,148.856
C03397=1122.205,-98.315,-46.413,179.616,4.474,148.857
C03398=1122.199,-98.065,-46.422,179.616,4.479,148.858
C03399=1122.194,-97.815,-46.431,179.615,4.484,148.859
C03400=1122.189,-97.565,-46.440,179.615,4.489,148.860
C03401=1122.184,-97.315,-46.449,179.614,4.494,148.861
C03402=1122.178,-97.065,-46.459,179.614,4.499,148.863
C03403=1122.173,-96.816,-46.468,179.614,4.504,148.864
C03404=1122.168,-96.566,-46.477,179.613,4.509,148.865
C03405=1122.163,-96.316,-46.486,179.613,4.514,148.866
C03406=1122.157,-96.066,-46.495,179.613,4.519,148.867
C03407=1122.151,-95.817,-46.504,179.613,4.524,148.869
C03408=1122.146,-95.567,-46.513,179.612,4.529,148.870
C03409=1122.141,-95.318,-46.522,179.612,4.533,148.871
C03410=1122.135,-95.068,-46.532,179.612,4.538,148.872
C03411=1122.130,-94.818,-46.541,179.612,4.544,148.873
C03412=1122.125,-94.568,-46.550,179.611,4.548,148.874
C03413=1122.119,-94.318,-46.559,179.611,4.553,148.875
C03414=1122.114,-94.068,-46.569,179.609,4.558,148.877
C03415=1122.109,-93.819,-46.578,179.609,4.563,148.878
C03416=1122.103,-93.568,-46.587,179.608,4.567,148.879
C03417=1122.098,-93.319,-46.596,179.608,4.572,148.880
C03418=1122.093,-93.069,-46.605,179.607,4.577,148.882
C03419=1122.088,-92.819,-46.615,179.606,4.582,148.883
C03420=1122.082,-92.569,-46.624,179.605,4.586,148.884
C03421=1122.077,-92.319,-46.633,179.605,4.591,148.885
C03422=1122.072,-92.070,-46.643,179.604,4.596,148.887
C03423=1122.066,-91.820,-46.652,179.604,4.601,148.888
C03424=1122.061,-91.570,-46.661,179.603,4.605,148.889
C03425=1122.055,-91.320,-46.671,179.603,4.611,148.890
C03426=1122.050,-91.071,-46.680,179.602,4.615,148.892
C03427=1122.044,-90.822,-46.689,179.601,4.621,148.893
C03428=1122.038,-90.572,-46.698,179.600,4.625,148.894
C03429=1122.033,-90.322,-46.708,179.600,4.630,148.895
C03430=1122.028,-90.072,-46.717,179.599,4.634,148.897
C03431=1122.022,-89.822,-46.726,179.599,4.640,148.898
C03432=1122.018,-89.573,-46.736,179.598,4.644,148.899
C03433=1122.012,-89.323,-46.745,179.598,4.649,148.900
C03434=1122.007,-89.107,-46.753,179.597,4.653,148.901
C03435=1122.003,-88.891,-46.761,179.597,4.658,148.902
C03436=1121.998,-88.676,-46.769,179.596,4.662,148.903
C03437=1121.993,-88.460,-46.777,179.596,4.666,148.905
C03438=1121.989,-88.246,-46.786,179.595,4.670,148.906
C03439=1121.985,-88.030,-46.794,179.595,4.675,148.907
C03440=1121.981,-87.814,-46.802,179.595,4.679,148.908
C03441=1121.975,-87.599,-46.810,179.594,4.684,148.909
C03442=1121.970,-87.349,-46.820,179.594,4.689,148.910
C03443=1121.964,-87.099,-46.829,179.593,4.693,148.911
C03444=1121.959,-86.849,-46.838,179.593,4.698,148.912
C03445=1121.954,-86.600,-46.848,179.593,4.703,148.914
C03446=1121.949,-86.349,-46.857,179.592,4.708,148.915
C03447=1121.944,-86.100,-46.867,179.591,4.713,148.916
C03448=1121.938,-85.850,-46.877,179.591,4.718,148.917
C03449=1121.933,-85.601,-46.886,179.591,4.724,148.918
C03450=1121.927,-85.350,-46.896,179.590,4.728,148.920
C03451=1121.922,-85.101,-46.905,179.590,4.733,148.921
C03452=1121.917,-84.851,-46.915,179.590,4.738,148.922
C03453=1121.911,-84.601,-46.924,179.589,4.744,148.923
C03454=1121.906,-84.352,-46.934,179.588,4.748,148.925
C03455=1121.901,-84.102,-46.943,179.588,4.753,148.926
C03456=1121.895,-83.852,-46.953,179.588,4.758,148.927
C03457=1121.890,-83.602,-46.962,179.588,4.764,148.928
C03458=1121.884,-83.353,-46.972,179.588,4.769,148.929
C03459=1121.879,-83.103,-46.981,179.588,4.774,148.930
C03460=1121.874,-82.853,-46.992,179.587,4.779,148.932
C03461=1121.869,-82.603,-47.000,179.587,4.783,148.933
C03462=1121.863,-82.353,-47.011,179.586,4.789,148.934
C03463=1121.859,-82.104,-47.020,179.586,4.794,148.935
C03464=1121.853,-81.854,-47.030,179.586,4.799,148.937
C03465=1121.848,-81.605,-47.039,179.585,4.804,148.938
C03466=1121.842,-81.355,-47.049,179.585,4.810,148.939
C03467=1121.836,-81.105,-47.059,179.585,4.815,148.940
C03468=1121.832,-80.854,-47.068,179.585,4.820,148.941
C03469=1121.826,-80.605,-47.079,179.585,4.825,148.942
C03470=1121.821,-80.356,-47.088,179.585,4.830,148.944
C03471=1121.815,-80.106,-47.098,179.584,4.835,148.945
C03472=1121.810,-79.856,-47.107,179.584,4.841,148.946
C03473=1121.805,-79.606,-47.117,179.584,4.846,148.947
C03474=1121.799,-79.357,-47.127,179.584,4.851,148.948
C03475=1121.794,-79.107,-47.137,179.584,4.856,148.949
C03476=1121.789,-78.857,-47.146,179.584,4.861,148.951
C03477=1121.783,-78.607,-47.157,179.583,4.866,148.952
C03478=1121.778,-78.358,-47.166,179.583,4.872,148.953
C03479=1121.772,-78.108,-47.176,179.583,4.877,148.954
C03480=1121.767,-77.858,-47.186,179.583,4.882,148.955
C03481=1121.762,-77.609,-47.196,179.583,4.887,148.956
C03482=1121.757,-77.358,-47.205,179.583,4.892,148.958
C03483=1121.751,-77.108,-47.216,179.583,4.897,148.959
C03484=1121.746,-76.859,-47.225,179.583,4.903,148.960
C03485=1121.741,-76.610,-47.235,179.583,4.908,148.961
C03486=1121.735,-76.359,-47.245,179.583,4.913,148.962
C03487=1121.730,-76.110,-47.255,179.583,4.918,148.963
C03488=1121.725,-75.860,-47.265,179.583,4.924,148.964
C03489=1121.719,-75.610,-47.275,179.583,4.929,148.966
C03490=1121.715,-75.395,-47.283,179.583,4.933,148.966
C03491=1121.710,-75.180,-47.292,179.583,4.937,148.967
C03492=1121.706,-74.964,-47.300,179.583,4.942,148.968
C03493=1121.701,-74.749,-47.310,179.584,4.947,148.969
C03494=1121.697,-74.533,-47.318,179.583,4.951,148.970
C03495=1121.691,-74.318,-47.326,179.583,4.956,148.971
C03496=1121.687,-74.102,-47.336,179.584,4.961,148.972
C03497=1121.683,-73.887,-47.344,179.583,4.965,148.973
C03498=1121.677,-73.637,-47.354,179.583,4.970,148.974
C03499=1121.671,-73.388,-47.364,179.584,4.976,148.975
C03500=1121.667,-73.138,-47.374,179.584,4.981,148.976
C03501=1121.662,-72.888,-47.384,179.584,4.986,148.978
C03502=1121.656,-72.639,-47.395,179.584,4.991,148.979
C03503=1121.650,-72.389,-47.405,179.585,4.997,148.980
C03504=1121.645,-72.138,-47.415,179.584,5.002,148.981
C03505=1121.640,-71.889,-47.424,179.584,5.007,148.982
C03506=1121.635,-71.639,-47.434,179.585,5.012,148.983
C03507=1121.630,-71.389,-47.445,179.585,5.018,148.984
C03508=1121.624,-71.140,-47.455,179.585,5.023,148.985
C03509=1121.618,-70.890,-47.465,179.586,5.028,148.986
C03510=1121.613,-70.641,-47.476,179.586,5.033,148.987
C03511=1121.609,-70.391,-47.486,179.586,5.038,148.988
C03512=1121.603,-70.141,-47.496,179.587,5.044,148.989
C03513=1121.597,-69.892,-47.506,179.587,5.049,148.991
C03514=1121.592,-69.641,-47.517,179.587,5.054,148.991
C03515=1121.587,-69.392,-47.527,179.587,5.060,148.993
C03516=1121.581,-69.142,-47.537,179.588,5.065,148.994
C03517=1121.576,-68.892,-47.548,179.588,5.070,148.995
C03518=1121.571,-68.642,-47.558,179.589,5.076,148.996
C03519=1121.566,-68.393,-47.567,179.588,5.081,148.997
C03520=1121.561,-68.143,-47.578,179.589,5.086,148.998
C03521=1121.555,-67.893,-47.588,179.589,5.091,148.999
C03522=1121.550,-67.643,-47.599,179.590,5.096,149.000
C03523=1121.544,-67.394,-47.609,179.591,5.102,149.001
C03524=1121.539,-67.144,-47.619,179.591,5.107,149.002
C03525=1121.534,-66.894,-47.630,179.592,5.112,149.003
C03526=1121.529,-66.645,-47.641,179.591,5.118,149.004
C03527=1121.523,-66.395,-47.651,179.592,5.123,149.005
C03528=1121.518,-66.145,-47.661,179.593,5.128,149.006
C03529=1121.512,-65.896,-47.672,179.593,5.134,149.007
C03530=1121.507,-65.645,-47.682,179.594,5.139,149.008
C03531=1121.502,-65.396,-47.692,179.594,5.143,149.009
C03532=1121.497,-65.146,-47.704,179.594,5.149,149.010
C03533=1121.492,-64.897,-47.714,179.595,5.154,149.011
C03534=1121.486,-64.647,-47.724,179.596,5.160,149.012
C03535=1121.481,-64.397,-47.735,179.596,5.164,149.013
C03536=1121.475,-64.147,-47.745,179.597,5.170,149.014
C03537=1121.471,-63.898,-47.756,179.598,5.176,149.015
C03538=1121.465,-63.648,-47.766,179.598,5.181,149.016
C03539=1121.460,-63.398,-47.777,179.599,5.186,149.017
C03540=1121.454,-63.148,-47.787,179.599,5.191,149.018
C03541=1121.450,-62.899,-47.798,179.600,5.197,149.018
C03542=1121.444,-62.649,-47.809,179.601,5.201,149.019
C03543=1121.439,-62.399,-47.819,179.602,5.207,149.020
C03544=1121.434,-62.150,-47.830,179.602,5.212,149.021
C03545=1121.429,-61.900,-47.841,179.603,5.218,149.022
C03546=1121.424,-61.685,-47.850,179.603,5.222,149.023
C03547=1121.419,-61.469,-47.859,179.604,5.227,149.024
C03548=1121.414,-61.254,-47.868,179.605,5.231,149.025
C03549=1121.410,-61.038,-47.878,179.606,5.236,149.025
C03550=1121.406,-60.823,-47.886,179.606,5.240,149.026
C03551=1121.401,-60.608,-47.896,179.607,5.245,149.027
C03552=1121.397,-60.393,-47.906,179.607,5.249,149.028
C03553=1121.392,-60.177,-47.915,179.608,5.254,149.028
C03554=1121.387,-59.927,-47.925,179.608,5.258,149.030
C03555=1121.382,-59.678,-47.936,179.608,5.263,149.031
C03556=1121.377,-59.428,-47.947,179.607,5.267,149.032
C03557=1121.371,-59.178,-47.958,179.608,5.272,149.033
C03558=1121.366,-58.929,-47.969,179.607,5.276,149.034
C03559=1121.360,-58.679,-47.979,179.607,5.281,149.035
C03560=1121.356,-58.429,-47.991,179.607,5.286,149.036
C03561=1121.350,-58.180,-48.001,179.607,5.291,149.037
C03562=1121.345,-57.930,-48.012,179.606,5.296,149.038
C03563=1121.340,-57.680,-48.023,179.606,5.300,149.039
C03564=1121.334,-57.431,-48.034,179.606,5.305,149.040
C03565=1121.329,-57.180,-48.045,179.605,5.309,149.041
C03566=1121.324,-56.932,-48.056,179.606,5.314,149.042
C03567=1121.319,-56.681,-48.066,179.606,5.319,149.043
C03568=1121.313,-56.432,-48.078,179.606,5.323,149.044
C03569=1121.308,-56.182,-48.088,179.605,5.328,149.046
C03570=1121.303,-55.932,-48.100,179.605,5.332,149.047
C03571=1121.298,-55.683,-48.110,179.605,5.337,149.048
C03572=1121.292,-55.433,-48.122,179.604,5.342,149.049
C03573=1121.287,-55.183,-48.132,179.604,5.347,149.050
C03574=1121.282,-54.934,-48.143,179.605,5.351,149.051
C03575=1121.277,-54.684,-48.154,179.604,5.356,149.052
C03576=1121.271,-54.434,-48.165,179.604,5.361,149.053
C03577=1121.266,-54.184,-48.177,179.604,5.365,149.054
C03578=1121.261,-53.934,-48.187,179.604,5.370,149.055
C03579=1121.256,-53.685,-48.198,179.604,5.375,149.056
C03580=1121.250,-53.435,-48.209,179.603,5.379,149.057
C03581=1121.245,-53.186,-48.220,179.603,5.384,149.058
C03582=1121.240,-52.936,-48.231,179.603,5.389,149.060
C03583=1121.234,-52.686,-48.243,179.603,5.393,149.060
C03584=1121.229,-52.437,-48.254,179.602,5.398,149.062
C03585=1121.224,-52.187,-48.265,179.602,5.403,149.063
C03586=1121.219,-51.936,-48.276,179.602,5.408,149.064
C03587=1121.213,-51.688,-48.287,179.602,5.412,149.065
C03588=1121.208,-51.437,-48.297,179.602,5.417,149.066
C03589=1121.203,-51.187,-48.309,179.601,5.421,149.067
C03590=1121.198,-50.938,-48.320,179.602,5.426,149.068
C03591=1121.193,-50.689,-48.332,179.602,5.431,149.069
C03592=1121.187,-50.438,-48.343,179.601,5.436,149.070
C03593=1121.182,-50.189,-48.354,179.601,5.440,149.071
C03594=1121.177,-49.940,-48.365,179.601,5.445,149.072
C03595=1121.172,-49.689,-48.376,179.601,5.450,149.074
C03596=1121.166,-49.440,-48.387,179.600,5.454,149.075
C03597=1121.162,-49.191,-48.398,179.600,5.459,149.076
C03598=1121.156,-48.940,-48.410,179.600,5.464,149.077
C03599=1121.151,-48.691,-48.420,179.600,5.468,149.078
C03600=1121.145,-48.441,-48.432,179.600,5.473,149.079
C03601=1121.140,-48.192,-48.444,179.599,5.478,149.080
C03602=1121.136,-47.976,-48.453,179.600,5.482,149.081
C03603=1121.131,-47.761,-48.463,179.600,5.486,149.082
C03604=1121.127,-47.546,-48.472,179.599,5.490,149.083
C03605=1121.122,-47.331,-48.482,179.599,5.494,149.084
C03606=1121.118,-47.115,-48.491,179.599,5.498,149.085
C03607=1121.113,-46.900,-48.502,179.599,5.502,149.085
C03608=1121.108,-46.685,-48.511,179.598,5.506,149.087
C03609=1121.104,-46.470,-48.521,179.598,5.510,149.087
C03610=1121.099,-46.220,-48.533,179.599,5.515,149.088
C03611=1121.093,-45.970,-48.544,179.598,5.519,149.090
C03612=1121.088,-45.721,-48.555,179.598,5.525,149.091
C03613=1121.083,-45.471,-48.567,179.598,5.530,149.092
C03614=1121.078,-45.221,-48.578,179.598,5.534,149.093
C03615=1121.072,-44.971,-48.590,179.597,5.539,149.094
C03616=1121.067,-44.722,-48.601,179.597,5.543,149.095
C03617=1121.062,-44.473,-48.612,179.597,5.548,149.096
C03618=1121.057,-44.222,-48.623,179.597,5.553,149.097
C03619=1121.052,-43.972,-48.635,179.597,5.557,149.098
C03620=1121.046,-43.723,-48.646,179.596,5.563,149.099
C03621=1121.041,-43.474,-48.657,179.596,5.566,149.100
C03622=1121.036,-43.224,-48.669,179.596,5.572,149.101
C03623=1121.031,-42.974,-48.680,179.596,5.577,149.103
C03624=1121.026,-42.724,-48.692,179.598,5.582,149.103
C03625=1121.020,-42.475,-48.704,179.600,5.588,149.104
C03626=1121.015,-42.225,-48.715,179.601,5.593,149.105
C03627=1121.010,-41.975,-48.727,179.602,5.599,149.105
C03628=1121.005,-41.726,-48.738,179.604,5.605,149.106
C03629=1121.000,-41.476,-48.750,179.606,5.610,149.107
